// TIA Portal V19 export
FUNCTION "ALARM" : Void   // FC6, LAD
{ S7_Optimized_Access := 'TRUE' }
// stored: SetENOAutomatically false
   VAR_TEMP
      QQ : Bool;
   END_VAR
   VAR_TEMP   // added for the SCL form of the ladder/FBD networks
      _w1 : Bool;
   END_VAR
BEGIN

REGION Network 1: ALARM RESET (MASTER TO SLAVE)
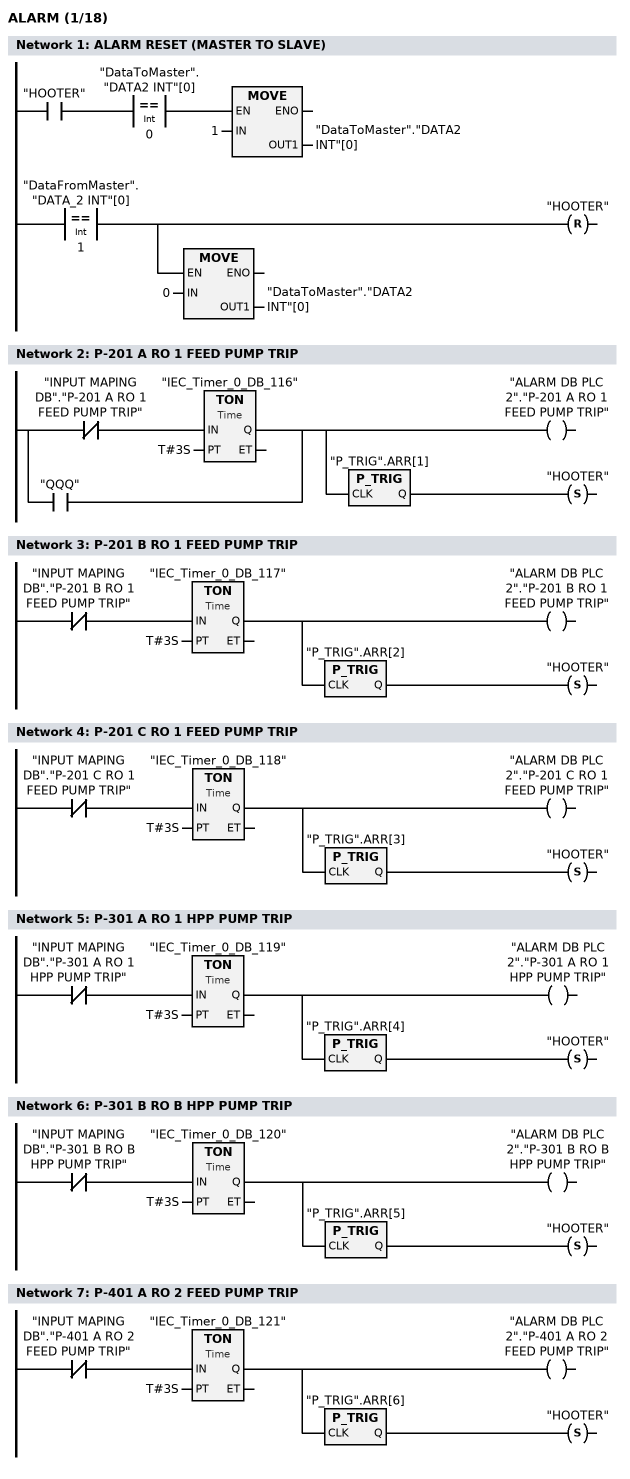
   RUNG wire#powerrail
      Contact( "HOOTER" )
      { S7_Templates := "SrcType := Int" } EQ_Contact(in1 := "DataToMaster"."DATA2 INT"[0], in2 := 0)
      Move(in := 1, out1 => "DataToMaster"."DATA2 INT"[0])
   END_RUNG
   RUNG wire#powerrail
      { S7_Templates := "SrcType := Int" } EQ_Contact(in1 := "DataFromMaster"."DATA_2 INT"[0], in2 := 1)
      wire#w1
      R_Coil( "HOOTER" )
   END_RUNG
   RUNG wire#w1
      Move(in := 0, out1 => "DataToMaster"."DATA2 INT"[0])
   END_RUNG
   // the same network as SCL:
   IF "HOOTER" AND ("DataToMaster"."DATA2 INT"[0] = 0) THEN "DataToMaster"."DATA2 INT"[0] := 1; END_IF;
   IF "DataFromMaster"."DATA_2 INT"[0] = 1 THEN
       "HOOTER" := FALSE;
       "DataToMaster"."DATA2 INT"[0] := 0;
   END_IF;
END_REGION

REGION Network 2: P-201 A RO 1 FEED PUMP TRIP
   RUNG wire#powerrail
      I_Contact( "INPUT MAPING DB"."P-201 A RO 1 FEED PUMP TRIP" )
      { S7_Templates := "time_type := Time" } "IEC_Timer_0_DB_116".TON(pt := T#3S, et =>)
      wire#w1
      Coil( "ALARM DB PLC 2"."P-201 A RO 1 FEED PUMP TRIP" )
   END_RUNG
   RUNG wire#powerrail
      Contact( "QQQ" )
   END_RUNG wire#w1
   RUNG wire#w1
      P_Trig( "P_TRIG".ARR[1] )
      S_Coil( "HOOTER" )
   END_RUNG
   // the same network as SCL:
   "IEC_Timer_0_DB_116".TON(IN := NOT "INPUT MAPING DB"."P-201 A RO 1 FEED PUMP TRIP", PT := T#3S);
   "ALARM DB PLC 2"."P-201 A RO 1 FEED PUMP TRIP" := "IEC_Timer_0_DB_116".Q OR "QQQ";
   #_w1 := "ALARM DB PLC 2"."P-201 A RO 1 FEED PUMP TRIP" AND NOT "P_TRIG".ARR[1];   // rising edge
   "P_TRIG".ARR[1] := "ALARM DB PLC 2"."P-201 A RO 1 FEED PUMP TRIP";
   IF #_w1 THEN "HOOTER" := TRUE; END_IF;
END_REGION

REGION Network 3: P-201 B RO 1 FEED PUMP TRIP
   RUNG wire#powerrail
      I_Contact( "INPUT MAPING DB"."P-201 B RO 1 FEED PUMP TRIP" )
      { S7_Templates := "time_type := Time" } "IEC_Timer_0_DB_117".TON(pt := T#3S, et =>)
      wire#w1
      Coil( "ALARM DB PLC 2"."P-201 B RO 1 FEED PUMP TRIP" )
   END_RUNG
   RUNG wire#w1
      P_Trig( "P_TRIG".ARR[2] )
      S_Coil( "HOOTER" )
   END_RUNG
   // the same network as SCL:
   "IEC_Timer_0_DB_117".TON(IN := NOT "INPUT MAPING DB"."P-201 B RO 1 FEED PUMP TRIP", PT := T#3S);
   "ALARM DB PLC 2"."P-201 B RO 1 FEED PUMP TRIP" := "IEC_Timer_0_DB_117".Q;
   #_w1 := "IEC_Timer_0_DB_117".Q AND NOT "P_TRIG".ARR[2];   // rising edge
   "P_TRIG".ARR[2] := "IEC_Timer_0_DB_117".Q;
   IF #_w1 THEN "HOOTER" := TRUE; END_IF;
END_REGION

REGION Network 4: P-201 C RO 1 FEED PUMP TRIP
   RUNG wire#powerrail
      I_Contact( "INPUT MAPING DB"."P-201 C RO 1 FEED PUMP TRIP" )
      { S7_Templates := "time_type := Time" } "IEC_Timer_0_DB_118".TON(pt := T#3S, et =>)
      wire#w1
      Coil( "ALARM DB PLC 2"."P-201 C RO 1 FEED PUMP TRIP" )
   END_RUNG
   RUNG wire#w1
      P_Trig( "P_TRIG".ARR[3] )
      S_Coil( "HOOTER" )
   END_RUNG
   // the same network as SCL:
   "IEC_Timer_0_DB_118".TON(IN := NOT "INPUT MAPING DB"."P-201 C RO 1 FEED PUMP TRIP", PT := T#3S);
   "ALARM DB PLC 2"."P-201 C RO 1 FEED PUMP TRIP" := "IEC_Timer_0_DB_118".Q;
   #_w1 := "IEC_Timer_0_DB_118".Q AND NOT "P_TRIG".ARR[3];   // rising edge
   "P_TRIG".ARR[3] := "IEC_Timer_0_DB_118".Q;
   IF #_w1 THEN "HOOTER" := TRUE; END_IF;
END_REGION

REGION Network 5: P-301 A RO 1 HPP PUMP TRIP
   RUNG wire#powerrail
      I_Contact( "INPUT MAPING DB"."P-301 A RO 1 HPP PUMP TRIP" )
      { S7_Templates := "time_type := Time" } "IEC_Timer_0_DB_119".TON(pt := T#3S, et =>)
      wire#w1
      Coil( "ALARM DB PLC 2"."P-301 A RO 1 HPP PUMP TRIP" )
   END_RUNG
   RUNG wire#w1
      P_Trig( "P_TRIG".ARR[4] )
      S_Coil( "HOOTER" )
   END_RUNG
   // the same network as SCL:
   "IEC_Timer_0_DB_119".TON(IN := NOT "INPUT MAPING DB"."P-301 A RO 1 HPP PUMP TRIP", PT := T#3S);
   "ALARM DB PLC 2"."P-301 A RO 1 HPP PUMP TRIP" := "IEC_Timer_0_DB_119".Q;
   #_w1 := "IEC_Timer_0_DB_119".Q AND NOT "P_TRIG".ARR[4];   // rising edge
   "P_TRIG".ARR[4] := "IEC_Timer_0_DB_119".Q;
   IF #_w1 THEN "HOOTER" := TRUE; END_IF;
END_REGION

REGION Network 6: P-301 B RO B HPP PUMP TRIP
   RUNG wire#powerrail
      I_Contact( "INPUT MAPING DB"."P-301 B RO B HPP PUMP TRIP" )
      { S7_Templates := "time_type := Time" } "IEC_Timer_0_DB_120".TON(pt := T#3S, et =>)
      wire#w1
      Coil( "ALARM DB PLC 2"."P-301 B RO B HPP PUMP TRIP" )
   END_RUNG
   RUNG wire#w1
      P_Trig( "P_TRIG".ARR[5] )
      S_Coil( "HOOTER" )
   END_RUNG
   // the same network as SCL:
   "IEC_Timer_0_DB_120".TON(IN := NOT "INPUT MAPING DB"."P-301 B RO B HPP PUMP TRIP", PT := T#3S);
   "ALARM DB PLC 2"."P-301 B RO B HPP PUMP TRIP" := "IEC_Timer_0_DB_120".Q;
   #_w1 := "IEC_Timer_0_DB_120".Q AND NOT "P_TRIG".ARR[5];   // rising edge
   "P_TRIG".ARR[5] := "IEC_Timer_0_DB_120".Q;
   IF #_w1 THEN "HOOTER" := TRUE; END_IF;
END_REGION

REGION Network 7: P-401 A RO 2 FEED PUMP TRIP
   RUNG wire#powerrail
      I_Contact( "INPUT MAPING DB"."P-401 A RO 2 FEED PUMP TRIP" )
      { S7_Templates := "time_type := Time" } "IEC_Timer_0_DB_121".TON(pt := T#3S, et =>)
      wire#w1
      Coil( "ALARM DB PLC 2"."P-401 A RO 2 FEED PUMP TRIP" )
   END_RUNG
   RUNG wire#w1
      P_Trig( "P_TRIG".ARR[6] )
      S_Coil( "HOOTER" )
   END_RUNG
   // the same network as SCL:
   "IEC_Timer_0_DB_121".TON(IN := NOT "INPUT MAPING DB"."P-401 A RO 2 FEED PUMP TRIP", PT := T#3S);
   "ALARM DB PLC 2"."P-401 A RO 2 FEED PUMP TRIP" := "IEC_Timer_0_DB_121".Q;
   #_w1 := "IEC_Timer_0_DB_121".Q AND NOT "P_TRIG".ARR[6];   // rising edge
   "P_TRIG".ARR[6] := "IEC_Timer_0_DB_121".Q;
   IF #_w1 THEN "HOOTER" := TRUE; END_IF;
END_REGION

REGION Network 8: P-401 B RO 2 FEED PUMP TRIP
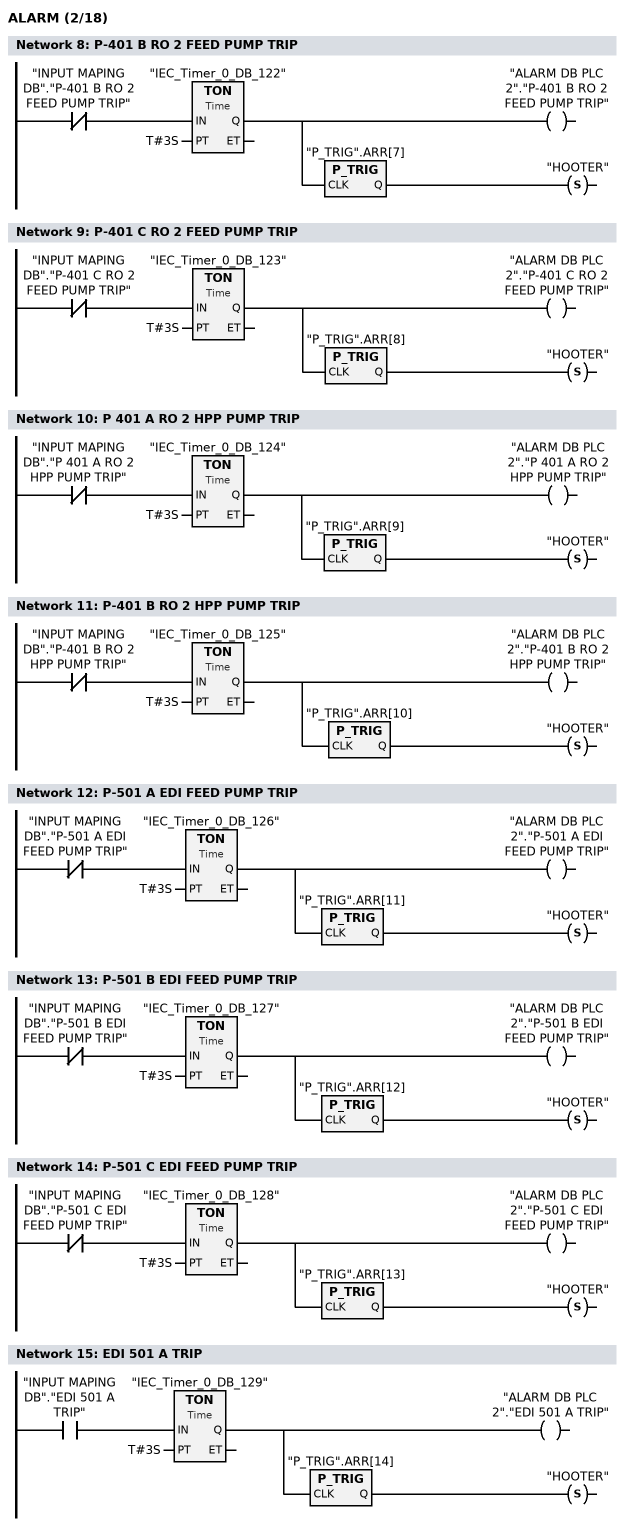
   RUNG wire#powerrail
      I_Contact( "INPUT MAPING DB"."P-401 B RO 2 FEED PUMP TRIP" )
      { S7_Templates := "time_type := Time" } "IEC_Timer_0_DB_122".TON(pt := T#3S, et =>)
      wire#w1
      Coil( "ALARM DB PLC 2"."P-401 B RO 2 FEED PUMP TRIP" )
   END_RUNG
   RUNG wire#w1
      P_Trig( "P_TRIG".ARR[7] )
      S_Coil( "HOOTER" )
   END_RUNG
   // the same network as SCL:
   "IEC_Timer_0_DB_122".TON(IN := NOT "INPUT MAPING DB"."P-401 B RO 2 FEED PUMP TRIP", PT := T#3S);
   "ALARM DB PLC 2"."P-401 B RO 2 FEED PUMP TRIP" := "IEC_Timer_0_DB_122".Q;
   #_w1 := "IEC_Timer_0_DB_122".Q AND NOT "P_TRIG".ARR[7];   // rising edge
   "P_TRIG".ARR[7] := "IEC_Timer_0_DB_122".Q;
   IF #_w1 THEN "HOOTER" := TRUE; END_IF;
END_REGION

REGION Network 9: P-401 C RO 2 FEED PUMP TRIP
   RUNG wire#powerrail
      I_Contact( "INPUT MAPING DB"."P-401 C RO 2 FEED PUMP TRIP" )
      { S7_Templates := "time_type := Time" } "IEC_Timer_0_DB_123".TON(pt := T#3S, et =>)
      wire#w1
      Coil( "ALARM DB PLC 2"."P-401 C RO 2 FEED PUMP TRIP" )
   END_RUNG
   RUNG wire#w1
      P_Trig( "P_TRIG".ARR[8] )
      S_Coil( "HOOTER" )
   END_RUNG
   // the same network as SCL:
   "IEC_Timer_0_DB_123".TON(IN := NOT "INPUT MAPING DB"."P-401 C RO 2 FEED PUMP TRIP", PT := T#3S);
   "ALARM DB PLC 2"."P-401 C RO 2 FEED PUMP TRIP" := "IEC_Timer_0_DB_123".Q;
   #_w1 := "IEC_Timer_0_DB_123".Q AND NOT "P_TRIG".ARR[8];   // rising edge
   "P_TRIG".ARR[8] := "IEC_Timer_0_DB_123".Q;
   IF #_w1 THEN "HOOTER" := TRUE; END_IF;
END_REGION

REGION Network 10: P 401 A RO 2 HPP PUMP TRIP
   RUNG wire#powerrail
      I_Contact( "INPUT MAPING DB"."P 401 A RO 2 HPP PUMP TRIP" )
      { S7_Templates := "time_type := Time" } "IEC_Timer_0_DB_124".TON(pt := T#3S, et =>)
      wire#w1
      Coil( "ALARM DB PLC 2"."P 401 A RO 2 HPP PUMP TRIP" )
   END_RUNG
   RUNG wire#w1
      P_Trig( "P_TRIG".ARR[9] )
      S_Coil( "HOOTER" )
   END_RUNG
   // the same network as SCL:
   "IEC_Timer_0_DB_124".TON(IN := NOT "INPUT MAPING DB"."P 401 A RO 2 HPP PUMP TRIP", PT := T#3S);
   "ALARM DB PLC 2"."P 401 A RO 2 HPP PUMP TRIP" := "IEC_Timer_0_DB_124".Q;
   #_w1 := "IEC_Timer_0_DB_124".Q AND NOT "P_TRIG".ARR[9];   // rising edge
   "P_TRIG".ARR[9] := "IEC_Timer_0_DB_124".Q;
   IF #_w1 THEN "HOOTER" := TRUE; END_IF;
END_REGION

REGION Network 11: P-401 B RO 2 HPP PUMP TRIP
   RUNG wire#powerrail
      I_Contact( "INPUT MAPING DB"."P-401 B RO 2 HPP PUMP TRIP" )
      { S7_Templates := "time_type := Time" } "IEC_Timer_0_DB_125".TON(pt := T#3S, et =>)
      wire#w1
      Coil( "ALARM DB PLC 2"."P-401 B RO 2 HPP PUMP TRIP" )
   END_RUNG
   RUNG wire#w1
      P_Trig( "P_TRIG".ARR[10] )
      S_Coil( "HOOTER" )
   END_RUNG
   // the same network as SCL:
   "IEC_Timer_0_DB_125".TON(IN := NOT "INPUT MAPING DB"."P-401 B RO 2 HPP PUMP TRIP", PT := T#3S);
   "ALARM DB PLC 2"."P-401 B RO 2 HPP PUMP TRIP" := "IEC_Timer_0_DB_125".Q;
   #_w1 := "IEC_Timer_0_DB_125".Q AND NOT "P_TRIG".ARR[10];   // rising edge
   "P_TRIG".ARR[10] := "IEC_Timer_0_DB_125".Q;
   IF #_w1 THEN "HOOTER" := TRUE; END_IF;
END_REGION

REGION Network 12: P-501 A EDI FEED PUMP TRIP
   RUNG wire#powerrail
      I_Contact( "INPUT MAPING DB"."P-501 A EDI FEED PUMP TRIP" )
      { S7_Templates := "time_type := Time" } "IEC_Timer_0_DB_126".TON(pt := T#3S, et =>)
      wire#w1
      Coil( "ALARM DB PLC 2"."P-501 A EDI FEED PUMP TRIP" )
   END_RUNG
   RUNG wire#w1
      P_Trig( "P_TRIG".ARR[11] )
      S_Coil( "HOOTER" )
   END_RUNG
   // the same network as SCL:
   "IEC_Timer_0_DB_126".TON(IN := NOT "INPUT MAPING DB"."P-501 A EDI FEED PUMP TRIP", PT := T#3S);
   "ALARM DB PLC 2"."P-501 A EDI FEED PUMP TRIP" := "IEC_Timer_0_DB_126".Q;
   #_w1 := "IEC_Timer_0_DB_126".Q AND NOT "P_TRIG".ARR[11];   // rising edge
   "P_TRIG".ARR[11] := "IEC_Timer_0_DB_126".Q;
   IF #_w1 THEN "HOOTER" := TRUE; END_IF;
END_REGION

REGION Network 13: P-501 B EDI FEED PUMP TRIP
   RUNG wire#powerrail
      I_Contact( "INPUT MAPING DB"."P-501 B EDI FEED PUMP TRIP" )
      { S7_Templates := "time_type := Time" } "IEC_Timer_0_DB_127".TON(pt := T#3S, et =>)
      wire#w1
      Coil( "ALARM DB PLC 2"."P-501 B EDI FEED PUMP TRIP" )
   END_RUNG
   RUNG wire#w1
      P_Trig( "P_TRIG".ARR[12] )
      S_Coil( "HOOTER" )
   END_RUNG
   // the same network as SCL:
   "IEC_Timer_0_DB_127".TON(IN := NOT "INPUT MAPING DB"."P-501 B EDI FEED PUMP TRIP", PT := T#3S);
   "ALARM DB PLC 2"."P-501 B EDI FEED PUMP TRIP" := "IEC_Timer_0_DB_127".Q;
   #_w1 := "IEC_Timer_0_DB_127".Q AND NOT "P_TRIG".ARR[12];   // rising edge
   "P_TRIG".ARR[12] := "IEC_Timer_0_DB_127".Q;
   IF #_w1 THEN "HOOTER" := TRUE; END_IF;
END_REGION

REGION Network 14: P-501 C EDI FEED PUMP TRIP
   RUNG wire#powerrail
      I_Contact( "INPUT MAPING DB"."P-501 C EDI FEED PUMP TRIP" )
      { S7_Templates := "time_type := Time" } "IEC_Timer_0_DB_128".TON(pt := T#3S, et =>)
      wire#w1
      Coil( "ALARM DB PLC 2"."P-501 C EDI FEED PUMP TRIP" )
   END_RUNG
   RUNG wire#w1
      P_Trig( "P_TRIG".ARR[13] )
      S_Coil( "HOOTER" )
   END_RUNG
   // the same network as SCL:
   "IEC_Timer_0_DB_128".TON(IN := NOT "INPUT MAPING DB"."P-501 C EDI FEED PUMP TRIP", PT := T#3S);
   "ALARM DB PLC 2"."P-501 C EDI FEED PUMP TRIP" := "IEC_Timer_0_DB_128".Q;
   #_w1 := "IEC_Timer_0_DB_128".Q AND NOT "P_TRIG".ARR[13];   // rising edge
   "P_TRIG".ARR[13] := "IEC_Timer_0_DB_128".Q;
   IF #_w1 THEN "HOOTER" := TRUE; END_IF;
END_REGION

REGION Network 15: EDI 501 A TRIP
   RUNG wire#powerrail
      Contact( "INPUT MAPING DB"."EDI 501 A TRIP" )
      { S7_Templates := "time_type := Time" } "IEC_Timer_0_DB_129".TON(pt := T#3S, et =>)
      wire#w1
      Coil( "ALARM DB PLC 2"."EDI 501 A TRIP" )
   END_RUNG
   RUNG wire#w1
      P_Trig( "P_TRIG".ARR[14] )
      S_Coil( "HOOTER" )
   END_RUNG
   // the same network as SCL:
   "IEC_Timer_0_DB_129".TON(IN := "INPUT MAPING DB"."EDI 501 A TRIP", PT := T#3S);
   "ALARM DB PLC 2"."EDI 501 A TRIP" := "IEC_Timer_0_DB_129".Q;
   #_w1 := "IEC_Timer_0_DB_129".Q AND NOT "P_TRIG".ARR[14];   // rising edge
   "P_TRIG".ARR[14] := "IEC_Timer_0_DB_129".Q;
   IF #_w1 THEN "HOOTER" := TRUE; END_IF;
END_REGION

REGION Network 16: EDI 501 B TRIP
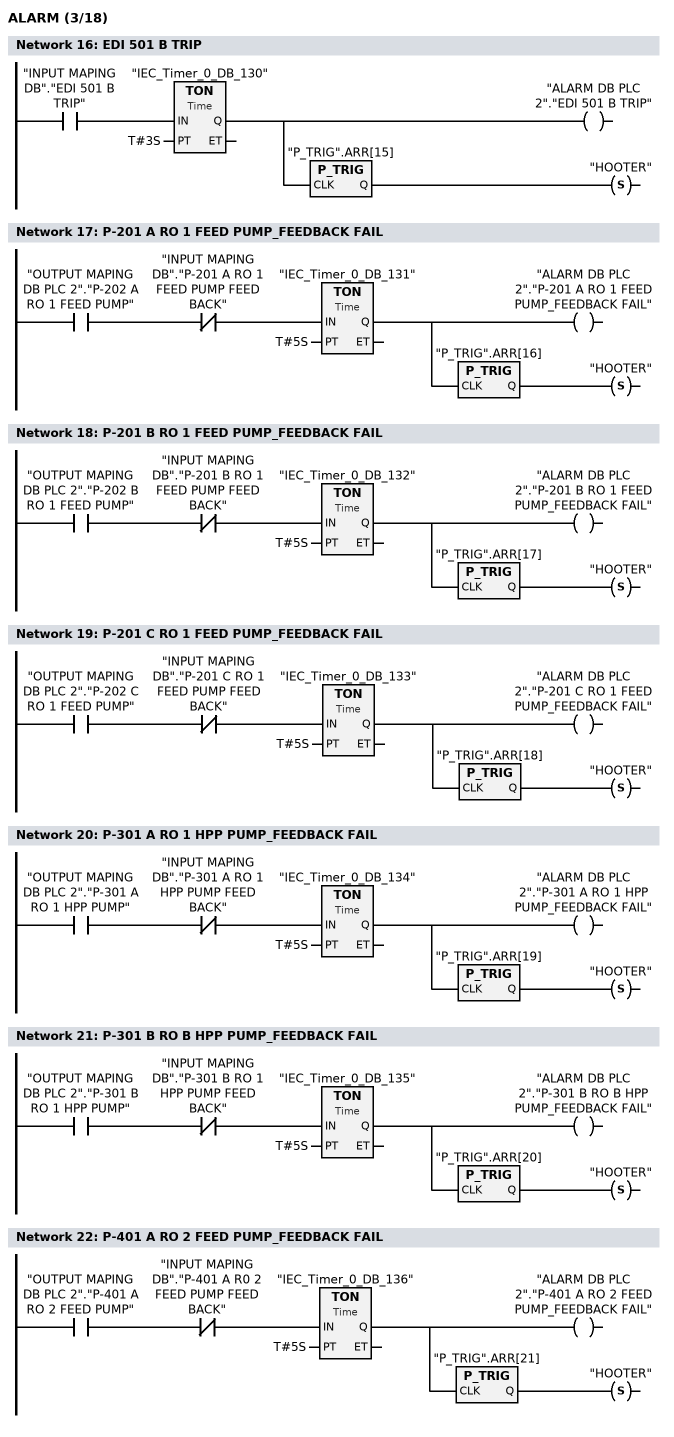
   RUNG wire#powerrail
      Contact( "INPUT MAPING DB"."EDI 501 B TRIP" )
      { S7_Templates := "time_type := Time" } "IEC_Timer_0_DB_130".TON(pt := T#3S, et =>)
      wire#w1
      Coil( "ALARM DB PLC 2"."EDI 501 B TRIP" )
   END_RUNG
   RUNG wire#w1
      P_Trig( "P_TRIG".ARR[15] )
      S_Coil( "HOOTER" )
   END_RUNG
   // the same network as SCL:
   "IEC_Timer_0_DB_130".TON(IN := "INPUT MAPING DB"."EDI 501 B TRIP", PT := T#3S);
   "ALARM DB PLC 2"."EDI 501 B TRIP" := "IEC_Timer_0_DB_130".Q;
   #_w1 := "IEC_Timer_0_DB_130".Q AND NOT "P_TRIG".ARR[15];   // rising edge
   "P_TRIG".ARR[15] := "IEC_Timer_0_DB_130".Q;
   IF #_w1 THEN "HOOTER" := TRUE; END_IF;
END_REGION

REGION Network 17: P-201 A RO 1 FEED PUMP_FEEDBACK FAIL
   RUNG wire#powerrail
      Contact( "OUTPUT MAPING DB PLC 2"."P-202 A RO 1 FEED PUMP" )
      I_Contact( "INPUT MAPING DB"."P-201 A RO 1 FEED PUMP FEED BACK" )
      { S7_Templates := "time_type := Time" } "IEC_Timer_0_DB_131".TON(pt := T#5S, et =>)
      wire#w1
      Coil( "ALARM DB PLC 2"."P-201 A RO 1 FEED PUMP_FEEDBACK FAIL" )
   END_RUNG
   RUNG wire#w1
      P_Trig( "P_TRIG".ARR[16] )
      S_Coil( "HOOTER" )
   END_RUNG
   // the same network as SCL:
   "IEC_Timer_0_DB_131".TON(IN := "OUTPUT MAPING DB PLC 2"."P-202 A RO 1 FEED PUMP" AND NOT "INPUT MAPING DB"."P-201 A RO 1 FEED PUMP FEED BACK",
                           PT := T#5S);
   "ALARM DB PLC 2"."P-201 A RO 1 FEED PUMP_FEEDBACK FAIL" := "IEC_Timer_0_DB_131".Q;
   #_w1 := "IEC_Timer_0_DB_131".Q AND NOT "P_TRIG".ARR[16];   // rising edge
   "P_TRIG".ARR[16] := "IEC_Timer_0_DB_131".Q;
   IF #_w1 THEN "HOOTER" := TRUE; END_IF;
END_REGION

REGION Network 18: P-201 B RO 1 FEED PUMP_FEEDBACK FAIL
   RUNG wire#powerrail
      Contact( "OUTPUT MAPING DB PLC 2"."P-202 B RO 1 FEED PUMP" )
      I_Contact( "INPUT MAPING DB"."P-201 B RO 1 FEED PUMP FEED BACK" )
      { S7_Templates := "time_type := Time" } "IEC_Timer_0_DB_132".TON(pt := T#5S, et =>)
      wire#w1
      Coil( "ALARM DB PLC 2"."P-201 B RO 1 FEED PUMP_FEEDBACK FAIL" )
   END_RUNG
   RUNG wire#w1
      P_Trig( "P_TRIG".ARR[17] )
      S_Coil( "HOOTER" )
   END_RUNG
   // the same network as SCL:
   "IEC_Timer_0_DB_132".TON(IN := "OUTPUT MAPING DB PLC 2"."P-202 B RO 1 FEED PUMP" AND NOT "INPUT MAPING DB"."P-201 B RO 1 FEED PUMP FEED BACK",
                           PT := T#5S);
   "ALARM DB PLC 2"."P-201 B RO 1 FEED PUMP_FEEDBACK FAIL" := "IEC_Timer_0_DB_132".Q;
   #_w1 := "IEC_Timer_0_DB_132".Q AND NOT "P_TRIG".ARR[17];   // rising edge
   "P_TRIG".ARR[17] := "IEC_Timer_0_DB_132".Q;
   IF #_w1 THEN "HOOTER" := TRUE; END_IF;
END_REGION

REGION Network 19: P-201 C RO 1 FEED PUMP_FEEDBACK FAIL
   RUNG wire#powerrail
      Contact( "OUTPUT MAPING DB PLC 2"."P-202 C RO 1 FEED PUMP" )
      I_Contact( "INPUT MAPING DB"."P-201 C RO 1 FEED PUMP FEED BACK" )
      { S7_Templates := "time_type := Time" } "IEC_Timer_0_DB_133".TON(pt := T#5S, et =>)
      wire#w1
      Coil( "ALARM DB PLC 2"."P-201 C RO 1 FEED PUMP_FEEDBACK FAIL" )
   END_RUNG
   RUNG wire#w1
      P_Trig( "P_TRIG".ARR[18] )
      S_Coil( "HOOTER" )
   END_RUNG
   // the same network as SCL:
   "IEC_Timer_0_DB_133".TON(IN := "OUTPUT MAPING DB PLC 2"."P-202 C RO 1 FEED PUMP" AND NOT "INPUT MAPING DB"."P-201 C RO 1 FEED PUMP FEED BACK",
                           PT := T#5S);
   "ALARM DB PLC 2"."P-201 C RO 1 FEED PUMP_FEEDBACK FAIL" := "IEC_Timer_0_DB_133".Q;
   #_w1 := "IEC_Timer_0_DB_133".Q AND NOT "P_TRIG".ARR[18];   // rising edge
   "P_TRIG".ARR[18] := "IEC_Timer_0_DB_133".Q;
   IF #_w1 THEN "HOOTER" := TRUE; END_IF;
END_REGION

REGION Network 20: P-301 A RO 1 HPP PUMP_FEEDBACK FAIL
   RUNG wire#powerrail
      Contact( "OUTPUT MAPING DB PLC 2"."P-301 A RO 1 HPP PUMP" )
      I_Contact( "INPUT MAPING DB"."P-301 A RO 1 HPP PUMP FEED BACK" )
      { S7_Templates := "time_type := Time" } "IEC_Timer_0_DB_134".TON(pt := T#5S, et =>)
      wire#w1
      Coil( "ALARM DB PLC 2"."P-301 A RO 1 HPP PUMP_FEEDBACK FAIL" )
   END_RUNG
   RUNG wire#w1
      P_Trig( "P_TRIG".ARR[19] )
      S_Coil( "HOOTER" )
   END_RUNG
   // the same network as SCL:
   "IEC_Timer_0_DB_134".TON(IN := "OUTPUT MAPING DB PLC 2"."P-301 A RO 1 HPP PUMP" AND NOT "INPUT MAPING DB"."P-301 A RO 1 HPP PUMP FEED BACK",
                           PT := T#5S);
   "ALARM DB PLC 2"."P-301 A RO 1 HPP PUMP_FEEDBACK FAIL" := "IEC_Timer_0_DB_134".Q;
   #_w1 := "IEC_Timer_0_DB_134".Q AND NOT "P_TRIG".ARR[19];   // rising edge
   "P_TRIG".ARR[19] := "IEC_Timer_0_DB_134".Q;
   IF #_w1 THEN "HOOTER" := TRUE; END_IF;
END_REGION

REGION Network 21: P-301 B RO B HPP PUMP_FEEDBACK FAIL
   RUNG wire#powerrail
      Contact( "OUTPUT MAPING DB PLC 2"."P-301 B RO 1 HPP PUMP" )
      I_Contact( "INPUT MAPING DB"."P-301 B RO 1 HPP PUMP FEED BACK" )
      { S7_Templates := "time_type := Time" } "IEC_Timer_0_DB_135".TON(pt := T#5S, et =>)
      wire#w1
      Coil( "ALARM DB PLC 2"."P-301 B RO B HPP PUMP_FEEDBACK FAIL" )
   END_RUNG
   RUNG wire#w1
      P_Trig( "P_TRIG".ARR[20] )
      S_Coil( "HOOTER" )
   END_RUNG
   // the same network as SCL:
   "IEC_Timer_0_DB_135".TON(IN := "OUTPUT MAPING DB PLC 2"."P-301 B RO 1 HPP PUMP" AND NOT "INPUT MAPING DB"."P-301 B RO 1 HPP PUMP FEED BACK",
                           PT := T#5S);
   "ALARM DB PLC 2"."P-301 B RO B HPP PUMP_FEEDBACK FAIL" := "IEC_Timer_0_DB_135".Q;
   #_w1 := "IEC_Timer_0_DB_135".Q AND NOT "P_TRIG".ARR[20];   // rising edge
   "P_TRIG".ARR[20] := "IEC_Timer_0_DB_135".Q;
   IF #_w1 THEN "HOOTER" := TRUE; END_IF;
END_REGION

REGION Network 22: P-401 A RO 2 FEED PUMP_FEEDBACK FAIL
   RUNG wire#powerrail
      Contact( "OUTPUT MAPING DB PLC 2"."P-401 A RO 2 FEED PUMP" )
      I_Contact( "INPUT MAPING DB"."P-401 A R0 2 FEED PUMP FEED BACK" )
      { S7_Templates := "time_type := Time" } "IEC_Timer_0_DB_136".TON(pt := T#5S, et =>)
      wire#w1
      Coil( "ALARM DB PLC 2"."P-401 A RO 2 FEED PUMP_FEEDBACK FAIL" )
   END_RUNG
   RUNG wire#w1
      P_Trig( "P_TRIG".ARR[21] )
      S_Coil( "HOOTER" )
   END_RUNG
   // the same network as SCL:
   "IEC_Timer_0_DB_136".TON(IN := "OUTPUT MAPING DB PLC 2"."P-401 A RO 2 FEED PUMP" AND NOT "INPUT MAPING DB"."P-401 A R0 2 FEED PUMP FEED BACK",
                           PT := T#5S);
   "ALARM DB PLC 2"."P-401 A RO 2 FEED PUMP_FEEDBACK FAIL" := "IEC_Timer_0_DB_136".Q;
   #_w1 := "IEC_Timer_0_DB_136".Q AND NOT "P_TRIG".ARR[21];   // rising edge
   "P_TRIG".ARR[21] := "IEC_Timer_0_DB_136".Q;
   IF #_w1 THEN "HOOTER" := TRUE; END_IF;
END_REGION

REGION Network 23: P-401 B RO 2 FEED PUMP_FEEDBACK FAIL
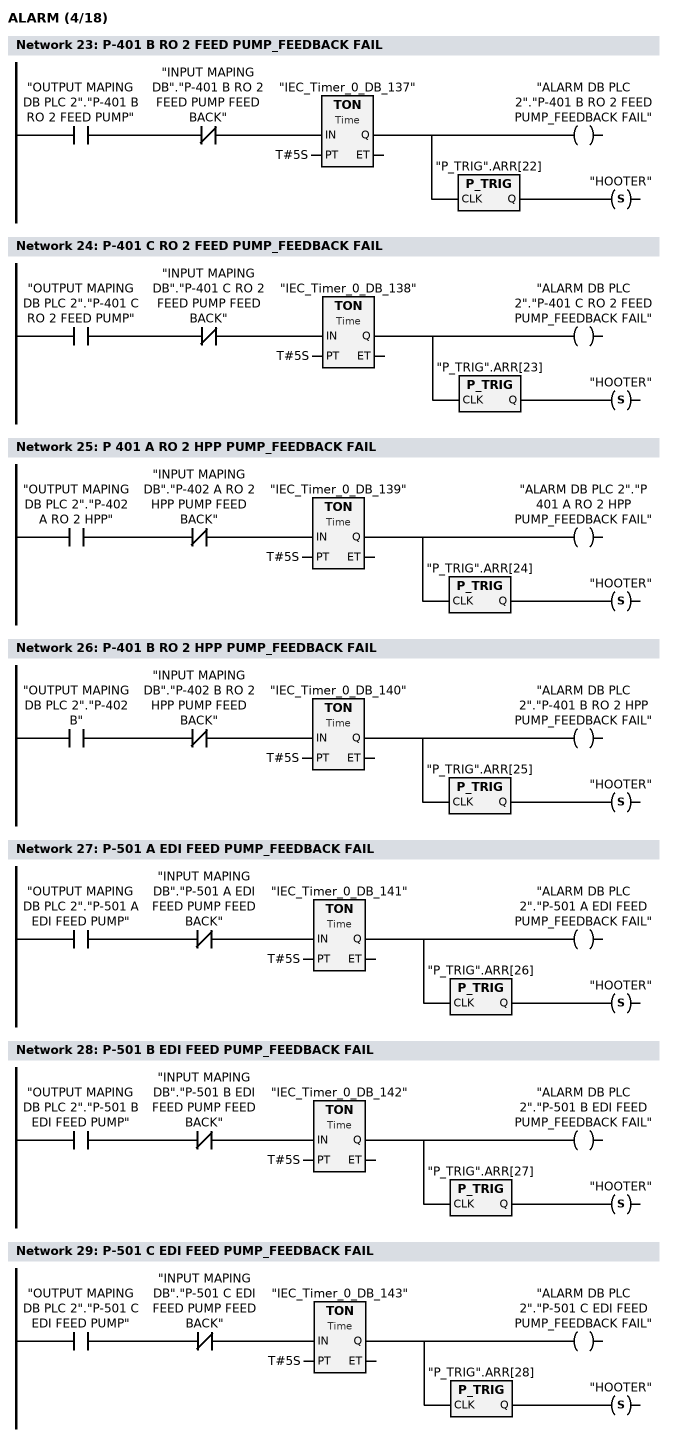
   RUNG wire#powerrail
      Contact( "OUTPUT MAPING DB PLC 2"."P-401 B RO 2 FEED PUMP" )
      I_Contact( "INPUT MAPING DB"."P-401 B RO 2 FEED PUMP FEED BACK" )
      { S7_Templates := "time_type := Time" } "IEC_Timer_0_DB_137".TON(pt := T#5S, et =>)
      wire#w1
      Coil( "ALARM DB PLC 2"."P-401 B RO 2 FEED PUMP_FEEDBACK FAIL" )
   END_RUNG
   RUNG wire#w1
      P_Trig( "P_TRIG".ARR[22] )
      S_Coil( "HOOTER" )
   END_RUNG
   // the same network as SCL:
   "IEC_Timer_0_DB_137".TON(IN := "OUTPUT MAPING DB PLC 2"."P-401 B RO 2 FEED PUMP" AND NOT "INPUT MAPING DB"."P-401 B RO 2 FEED PUMP FEED BACK",
                           PT := T#5S);
   "ALARM DB PLC 2"."P-401 B RO 2 FEED PUMP_FEEDBACK FAIL" := "IEC_Timer_0_DB_137".Q;
   #_w1 := "IEC_Timer_0_DB_137".Q AND NOT "P_TRIG".ARR[22];   // rising edge
   "P_TRIG".ARR[22] := "IEC_Timer_0_DB_137".Q;
   IF #_w1 THEN "HOOTER" := TRUE; END_IF;
END_REGION

REGION Network 24: P-401 C RO 2 FEED PUMP_FEEDBACK FAIL
   RUNG wire#powerrail
      Contact( "OUTPUT MAPING DB PLC 2"."P-401 C RO 2 FEED PUMP" )
      I_Contact( "INPUT MAPING DB"."P-401 C RO 2 FEED PUMP FEED BACK" )
      { S7_Templates := "time_type := Time" } "IEC_Timer_0_DB_138".TON(pt := T#5S, et =>)
      wire#w1
      Coil( "ALARM DB PLC 2"."P-401 C RO 2 FEED PUMP_FEEDBACK FAIL" )
   END_RUNG
   RUNG wire#w1
      P_Trig( "P_TRIG".ARR[23] )
      S_Coil( "HOOTER" )
   END_RUNG
   // the same network as SCL:
   "IEC_Timer_0_DB_138".TON(IN := "OUTPUT MAPING DB PLC 2"."P-401 C RO 2 FEED PUMP" AND NOT "INPUT MAPING DB"."P-401 C RO 2 FEED PUMP FEED BACK",
                           PT := T#5S);
   "ALARM DB PLC 2"."P-401 C RO 2 FEED PUMP_FEEDBACK FAIL" := "IEC_Timer_0_DB_138".Q;
   #_w1 := "IEC_Timer_0_DB_138".Q AND NOT "P_TRIG".ARR[23];   // rising edge
   "P_TRIG".ARR[23] := "IEC_Timer_0_DB_138".Q;
   IF #_w1 THEN "HOOTER" := TRUE; END_IF;
END_REGION

REGION Network 25: P 401 A RO 2 HPP PUMP_FEEDBACK FAIL
   RUNG wire#powerrail
      Contact( "OUTPUT MAPING DB PLC 2"."P-402  A RO 2 HPP" )
      I_Contact( "INPUT MAPING DB"."P-402 A RO 2 HPP PUMP FEED BACK" )
      { S7_Templates := "time_type := Time" } "IEC_Timer_0_DB_139".TON(pt := T#5S, et =>)
      wire#w1
      Coil( "ALARM DB PLC 2"."P 401 A RO 2 HPP PUMP_FEEDBACK FAIL" )
   END_RUNG
   RUNG wire#w1
      P_Trig( "P_TRIG".ARR[24] )
      S_Coil( "HOOTER" )
   END_RUNG
   // the same network as SCL:
   "IEC_Timer_0_DB_139".TON(IN := "OUTPUT MAPING DB PLC 2"."P-402  A RO 2 HPP" AND NOT "INPUT MAPING DB"."P-402 A RO 2 HPP PUMP FEED BACK",
                           PT := T#5S);
   "ALARM DB PLC 2"."P 401 A RO 2 HPP PUMP_FEEDBACK FAIL" := "IEC_Timer_0_DB_139".Q;
   #_w1 := "IEC_Timer_0_DB_139".Q AND NOT "P_TRIG".ARR[24];   // rising edge
   "P_TRIG".ARR[24] := "IEC_Timer_0_DB_139".Q;
   IF #_w1 THEN "HOOTER" := TRUE; END_IF;
END_REGION

REGION Network 26: P-401 B RO 2 HPP PUMP_FEEDBACK FAIL
   RUNG wire#powerrail
      Contact( "OUTPUT MAPING DB PLC 2"."P-402 B" )
      I_Contact( "INPUT MAPING DB"."P-402 B RO 2 HPP PUMP FEED BACK" )
      { S7_Templates := "time_type := Time" } "IEC_Timer_0_DB_140".TON(pt := T#5S, et =>)
      wire#w1
      Coil( "ALARM DB PLC 2"."P-401 B RO 2 HPP PUMP_FEEDBACK FAIL" )
   END_RUNG
   RUNG wire#w1
      P_Trig( "P_TRIG".ARR[25] )
      S_Coil( "HOOTER" )
   END_RUNG
   // the same network as SCL:
   "IEC_Timer_0_DB_140".TON(IN := "OUTPUT MAPING DB PLC 2"."P-402 B" AND NOT "INPUT MAPING DB"."P-402 B RO 2 HPP PUMP FEED BACK",
                           PT := T#5S);
   "ALARM DB PLC 2"."P-401 B RO 2 HPP PUMP_FEEDBACK FAIL" := "IEC_Timer_0_DB_140".Q;
   #_w1 := "IEC_Timer_0_DB_140".Q AND NOT "P_TRIG".ARR[25];   // rising edge
   "P_TRIG".ARR[25] := "IEC_Timer_0_DB_140".Q;
   IF #_w1 THEN "HOOTER" := TRUE; END_IF;
END_REGION

REGION Network 27: P-501 A EDI FEED PUMP_FEEDBACK FAIL
   RUNG wire#powerrail
      Contact( "OUTPUT MAPING DB PLC 2"."P-501 A EDI FEED PUMP" )
      I_Contact( "INPUT MAPING DB"."P-501 A EDI FEED PUMP FEED BACK" )
      { S7_Templates := "time_type := Time" } "IEC_Timer_0_DB_141".TON(pt := T#5S, et =>)
      wire#w1
      Coil( "ALARM DB PLC 2"."P-501 A EDI FEED PUMP_FEEDBACK FAIL" )
   END_RUNG
   RUNG wire#w1
      P_Trig( "P_TRIG".ARR[26] )
      S_Coil( "HOOTER" )
   END_RUNG
   // the same network as SCL:
   "IEC_Timer_0_DB_141".TON(IN := "OUTPUT MAPING DB PLC 2"."P-501 A EDI FEED PUMP" AND NOT "INPUT MAPING DB"."P-501 A EDI FEED PUMP FEED BACK",
                           PT := T#5S);
   "ALARM DB PLC 2"."P-501 A EDI FEED PUMP_FEEDBACK FAIL" := "IEC_Timer_0_DB_141".Q;
   #_w1 := "IEC_Timer_0_DB_141".Q AND NOT "P_TRIG".ARR[26];   // rising edge
   "P_TRIG".ARR[26] := "IEC_Timer_0_DB_141".Q;
   IF #_w1 THEN "HOOTER" := TRUE; END_IF;
END_REGION

REGION Network 28: P-501 B EDI FEED PUMP_FEEDBACK FAIL
   RUNG wire#powerrail
      Contact( "OUTPUT MAPING DB PLC 2"."P-501 B EDI FEED PUMP" )
      I_Contact( "INPUT MAPING DB"."P-501 B EDI FEED PUMP FEED BACK" )
      { S7_Templates := "time_type := Time" } "IEC_Timer_0_DB_142".TON(pt := T#5S, et =>)
      wire#w1
      Coil( "ALARM DB PLC 2"."P-501 B EDI FEED PUMP_FEEDBACK FAIL" )
   END_RUNG
   RUNG wire#w1
      P_Trig( "P_TRIG".ARR[27] )
      S_Coil( "HOOTER" )
   END_RUNG
   // the same network as SCL:
   "IEC_Timer_0_DB_142".TON(IN := "OUTPUT MAPING DB PLC 2"."P-501 B EDI FEED PUMP" AND NOT "INPUT MAPING DB"."P-501 B EDI FEED PUMP FEED BACK",
                           PT := T#5S);
   "ALARM DB PLC 2"."P-501 B EDI FEED PUMP_FEEDBACK FAIL" := "IEC_Timer_0_DB_142".Q;
   #_w1 := "IEC_Timer_0_DB_142".Q AND NOT "P_TRIG".ARR[27];   // rising edge
   "P_TRIG".ARR[27] := "IEC_Timer_0_DB_142".Q;
   IF #_w1 THEN "HOOTER" := TRUE; END_IF;
END_REGION

REGION Network 29: P-501 C EDI FEED PUMP_FEEDBACK FAIL
   RUNG wire#powerrail
      Contact( "OUTPUT MAPING DB PLC 2"."P-501 C EDI FEED PUMP" )
      I_Contact( "INPUT MAPING DB"."P-501 C EDI FEED PUMP FEED BACK" )
      { S7_Templates := "time_type := Time" } "IEC_Timer_0_DB_143".TON(pt := T#5S, et =>)
      wire#w1
      Coil( "ALARM DB PLC 2"."P-501 C EDI FEED PUMP_FEEDBACK FAIL" )
   END_RUNG
   RUNG wire#w1
      P_Trig( "P_TRIG".ARR[28] )
      S_Coil( "HOOTER" )
   END_RUNG
   // the same network as SCL:
   "IEC_Timer_0_DB_143".TON(IN := "OUTPUT MAPING DB PLC 2"."P-501 C EDI FEED PUMP" AND NOT "INPUT MAPING DB"."P-501 C EDI FEED PUMP FEED BACK",
                           PT := T#5S);
   "ALARM DB PLC 2"."P-501 C EDI FEED PUMP_FEEDBACK FAIL" := "IEC_Timer_0_DB_143".Q;
   #_w1 := "IEC_Timer_0_DB_143".Q AND NOT "P_TRIG".ARR[28];   // rising edge
   "P_TRIG".ARR[28] := "IEC_Timer_0_DB_143".Q;
   IF #_w1 THEN "HOOTER" := TRUE; END_IF;
END_REGION

REGION Network 30: EDI 501 A _FEEDBACK FAIL
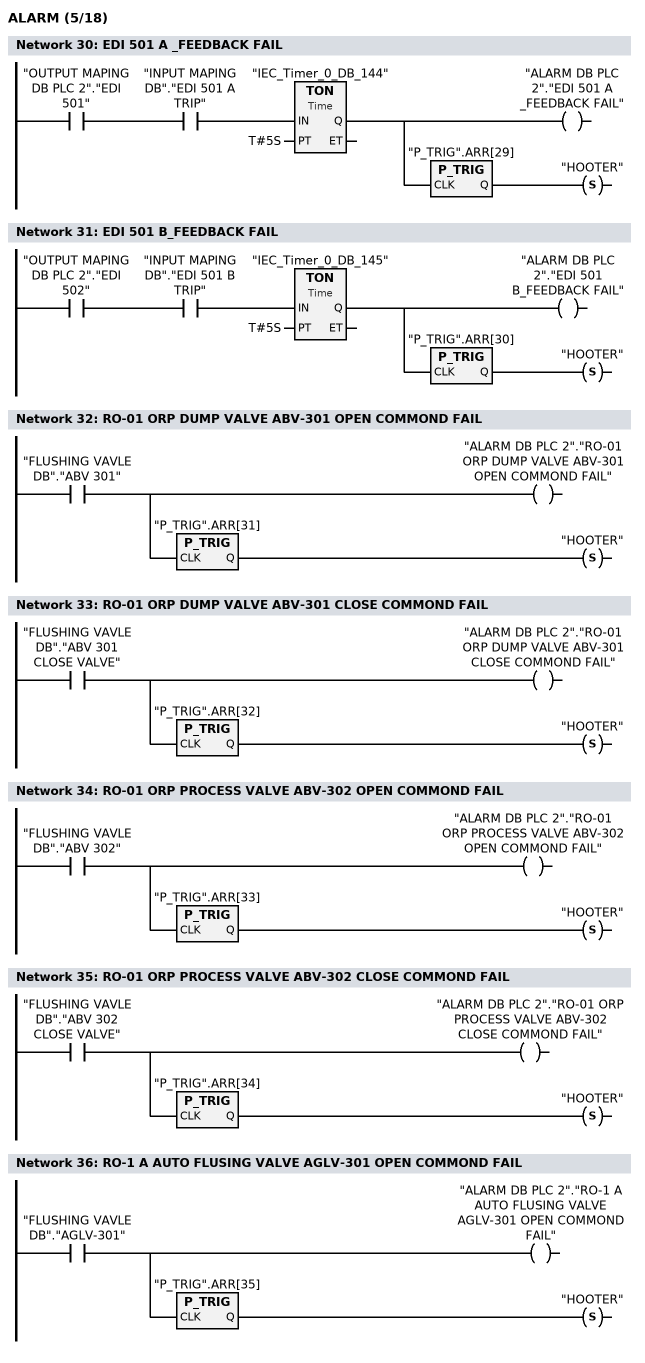
   RUNG wire#powerrail
      Contact( "OUTPUT MAPING DB PLC 2"."EDI 501" )
      Contact( "INPUT MAPING DB"."EDI 501 A TRIP" )
      { S7_Templates := "time_type := Time" } "IEC_Timer_0_DB_144".TON(pt := T#5S, et =>)
      wire#w1
      Coil( "ALARM DB PLC 2"."EDI 501 A _FEEDBACK FAIL" )
   END_RUNG
   RUNG wire#w1
      P_Trig( "P_TRIG".ARR[29] )
      S_Coil( "HOOTER" )
   END_RUNG
   // the same network as SCL:
   "IEC_Timer_0_DB_144".TON(IN := "OUTPUT MAPING DB PLC 2"."EDI 501" AND "INPUT MAPING DB"."EDI 501 A TRIP",
                           PT := T#5S);
   "ALARM DB PLC 2"."EDI 501 A _FEEDBACK FAIL" := "IEC_Timer_0_DB_144".Q;
   #_w1 := "IEC_Timer_0_DB_144".Q AND NOT "P_TRIG".ARR[29];   // rising edge
   "P_TRIG".ARR[29] := "IEC_Timer_0_DB_144".Q;
   IF #_w1 THEN "HOOTER" := TRUE; END_IF;
END_REGION

REGION Network 31: EDI 501 B_FEEDBACK FAIL
   RUNG wire#powerrail
      Contact( "OUTPUT MAPING DB PLC 2"."EDI 502" )
      Contact( "INPUT MAPING DB"."EDI 501 B TRIP" )
      { S7_Templates := "time_type := Time" } "IEC_Timer_0_DB_145".TON(pt := T#5S, et =>)
      wire#w1
      Coil( "ALARM DB PLC 2"."EDI 501 B_FEEDBACK FAIL" )
   END_RUNG
   RUNG wire#w1
      P_Trig( "P_TRIG".ARR[30] )
      S_Coil( "HOOTER" )
   END_RUNG
   // the same network as SCL:
   "IEC_Timer_0_DB_145".TON(IN := "OUTPUT MAPING DB PLC 2"."EDI 502" AND "INPUT MAPING DB"."EDI 501 B TRIP",
                           PT := T#5S);
   "ALARM DB PLC 2"."EDI 501 B_FEEDBACK FAIL" := "IEC_Timer_0_DB_145".Q;
   #_w1 := "IEC_Timer_0_DB_145".Q AND NOT "P_TRIG".ARR[30];   // rising edge
   "P_TRIG".ARR[30] := "IEC_Timer_0_DB_145".Q;
   IF #_w1 THEN "HOOTER" := TRUE; END_IF;
END_REGION

REGION Network 32: RO-01 ORP DUMP VALVE ABV-301 OPEN COMMOND FAIL
   RUNG wire#powerrail
      Contact( "FLUSHING VAVLE DB"."ABV 301" )
      wire#w1
      Coil( "ALARM DB PLC 2"."RO-01 ORP DUMP VALVE ABV-301 OPEN COMMOND FAIL" )
   END_RUNG
   RUNG wire#w1
      P_Trig( "P_TRIG".ARR[31] )
      S_Coil( "HOOTER" )
   END_RUNG
   // the same network as SCL:
   "ALARM DB PLC 2"."RO-01 ORP DUMP VALVE ABV-301 OPEN COMMOND FAIL" := "FLUSHING VAVLE DB"."ABV 301";
   #_w1 := "FLUSHING VAVLE DB"."ABV 301" AND NOT "P_TRIG".ARR[31];   // rising edge
   "P_TRIG".ARR[31] := "FLUSHING VAVLE DB"."ABV 301";
   IF #_w1 THEN "HOOTER" := TRUE; END_IF;
END_REGION

REGION Network 33: RO-01 ORP DUMP VALVE ABV-301 CLOSE COMMOND FAIL
   RUNG wire#powerrail
      Contact( "FLUSHING VAVLE DB"."ABV 301 CLOSE VALVE" )
      wire#w1
      Coil( "ALARM DB PLC 2"."RO-01 ORP DUMP VALVE ABV-301 CLOSE COMMOND FAIL" )
   END_RUNG
   RUNG wire#w1
      P_Trig( "P_TRIG".ARR[32] )
      S_Coil( "HOOTER" )
   END_RUNG
   // the same network as SCL:
   "ALARM DB PLC 2"."RO-01 ORP DUMP VALVE ABV-301 CLOSE COMMOND FAIL" := "FLUSHING VAVLE DB"."ABV 301 CLOSE VALVE";
   #_w1 := "FLUSHING VAVLE DB"."ABV 301 CLOSE VALVE" AND NOT "P_TRIG".ARR[32];   // rising edge
   "P_TRIG".ARR[32] := "FLUSHING VAVLE DB"."ABV 301 CLOSE VALVE";
   IF #_w1 THEN "HOOTER" := TRUE; END_IF;
END_REGION

REGION Network 34: RO-01 ORP PROCESS VALVE ABV-302 OPEN COMMOND FAIL
   RUNG wire#powerrail
      Contact( "FLUSHING VAVLE DB"."ABV 302" )
      wire#w1
      Coil( "ALARM DB PLC 2"."RO-01 ORP PROCESS VALVE ABV-302 OPEN COMMOND FAIL" )
   END_RUNG
   RUNG wire#w1
      P_Trig( "P_TRIG".ARR[33] )
      S_Coil( "HOOTER" )
   END_RUNG
   // the same network as SCL:
   "ALARM DB PLC 2"."RO-01 ORP PROCESS VALVE ABV-302 OPEN COMMOND FAIL" := "FLUSHING VAVLE DB"."ABV 302";
   #_w1 := "FLUSHING VAVLE DB"."ABV 302" AND NOT "P_TRIG".ARR[33];   // rising edge
   "P_TRIG".ARR[33] := "FLUSHING VAVLE DB"."ABV 302";
   IF #_w1 THEN "HOOTER" := TRUE; END_IF;
END_REGION

REGION Network 35: RO-01 ORP PROCESS VALVE ABV-302 CLOSE COMMOND FAIL
   RUNG wire#powerrail
      Contact( "FLUSHING VAVLE DB"."ABV 302 CLOSE VALVE" )
      wire#w1
      Coil( "ALARM DB PLC 2"."RO-01 ORP PROCESS VALVE ABV-302 CLOSE COMMOND FAIL" )
   END_RUNG
   RUNG wire#w1
      P_Trig( "P_TRIG".ARR[34] )
      S_Coil( "HOOTER" )
   END_RUNG
   // the same network as SCL:
   "ALARM DB PLC 2"."RO-01 ORP PROCESS VALVE ABV-302 CLOSE COMMOND FAIL" := "FLUSHING VAVLE DB"."ABV 302 CLOSE VALVE";
   #_w1 := "FLUSHING VAVLE DB"."ABV 302 CLOSE VALVE" AND NOT "P_TRIG".ARR[34];   // rising edge
   "P_TRIG".ARR[34] := "FLUSHING VAVLE DB"."ABV 302 CLOSE VALVE";
   IF #_w1 THEN "HOOTER" := TRUE; END_IF;
END_REGION

REGION Network 36: RO-1 A AUTO FLUSING VALVE AGLV-301 OPEN COMMOND FAIL
   RUNG wire#powerrail
      Contact( "FLUSHING VAVLE DB"."AGLV-301" )
      wire#w1
      Coil( "ALARM DB PLC 2"."RO-1 A AUTO FLUSING VALVE AGLV-301 OPEN COMMOND FAIL" )
   END_RUNG
   RUNG wire#w1
      P_Trig( "P_TRIG".ARR[35] )
      S_Coil( "HOOTER" )
   END_RUNG
   // the same network as SCL:
   "ALARM DB PLC 2"."RO-1 A AUTO FLUSING VALVE AGLV-301 OPEN COMMOND FAIL" := "FLUSHING VAVLE DB"."AGLV-301";
   #_w1 := "FLUSHING VAVLE DB"."AGLV-301" AND NOT "P_TRIG".ARR[35];   // rising edge
   "P_TRIG".ARR[35] := "FLUSHING VAVLE DB"."AGLV-301";
   IF #_w1 THEN "HOOTER" := TRUE; END_IF;
END_REGION

REGION Network 37: RO-1 A AUTO FLUSING VALVE AGLV-301 CLOSE COMMOND FAIL
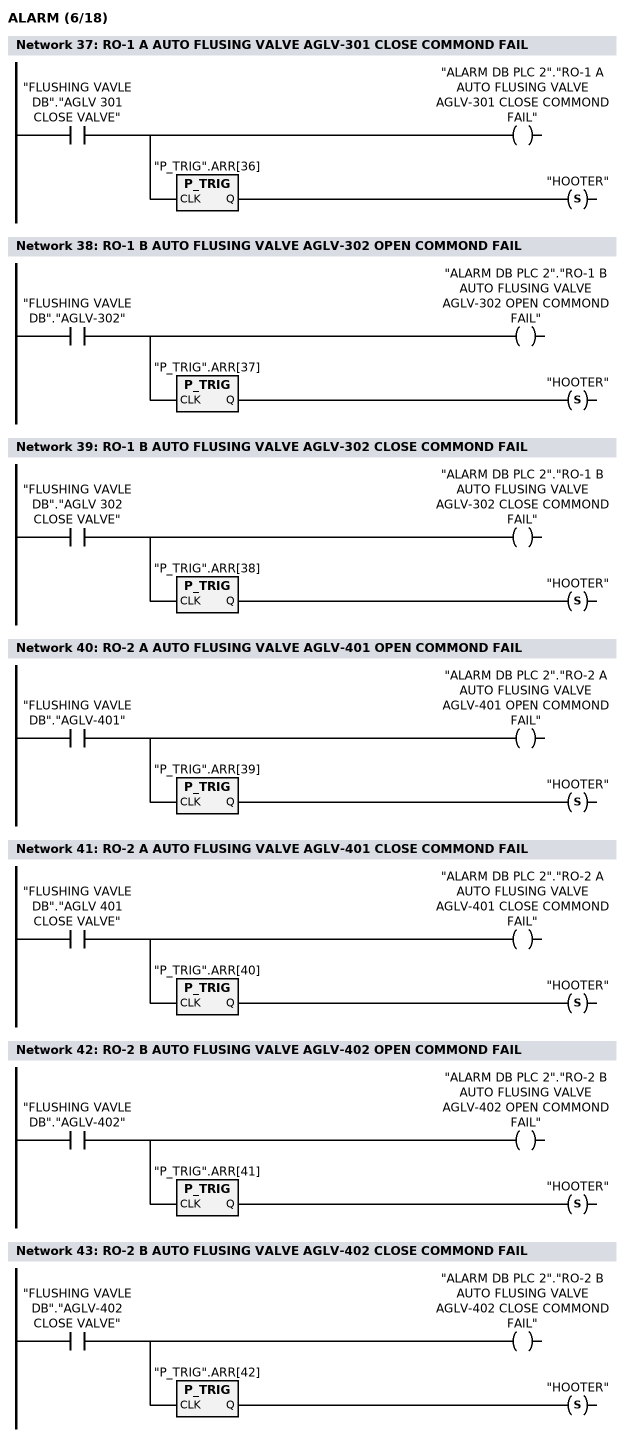
   RUNG wire#powerrail
      Contact( "FLUSHING VAVLE DB"."AGLV 301 CLOSE VALVE" )
      wire#w1
      Coil( "ALARM DB PLC 2"."RO-1 A AUTO FLUSING VALVE AGLV-301 CLOSE COMMOND FAIL" )
   END_RUNG
   RUNG wire#w1
      P_Trig( "P_TRIG".ARR[36] )
      S_Coil( "HOOTER" )
   END_RUNG
   // the same network as SCL:
   "ALARM DB PLC 2"."RO-1 A AUTO FLUSING VALVE AGLV-301 CLOSE COMMOND FAIL" := "FLUSHING VAVLE DB"."AGLV 301 CLOSE VALVE";
   #_w1 := "FLUSHING VAVLE DB"."AGLV 301 CLOSE VALVE" AND NOT "P_TRIG".ARR[36];   // rising edge
   "P_TRIG".ARR[36] := "FLUSHING VAVLE DB"."AGLV 301 CLOSE VALVE";
   IF #_w1 THEN "HOOTER" := TRUE; END_IF;
END_REGION

REGION Network 38: RO-1 B AUTO FLUSING VALVE AGLV-302 OPEN COMMOND FAIL
   RUNG wire#powerrail
      Contact( "FLUSHING VAVLE DB"."AGLV-302" )
      wire#w1
      Coil( "ALARM DB PLC 2"."RO-1 B AUTO FLUSING VALVE AGLV-302 OPEN COMMOND FAIL" )
   END_RUNG
   RUNG wire#w1
      P_Trig( "P_TRIG".ARR[37] )
      S_Coil( "HOOTER" )
   END_RUNG
   // the same network as SCL:
   "ALARM DB PLC 2"."RO-1 B AUTO FLUSING VALVE AGLV-302 OPEN COMMOND FAIL" := "FLUSHING VAVLE DB"."AGLV-302";
   #_w1 := "FLUSHING VAVLE DB"."AGLV-302" AND NOT "P_TRIG".ARR[37];   // rising edge
   "P_TRIG".ARR[37] := "FLUSHING VAVLE DB"."AGLV-302";
   IF #_w1 THEN "HOOTER" := TRUE; END_IF;
END_REGION

REGION Network 39: RO-1 B AUTO FLUSING VALVE AGLV-302 CLOSE COMMOND FAIL
   RUNG wire#powerrail
      Contact( "FLUSHING VAVLE DB"."AGLV 302 CLOSE VALVE" )
      wire#w1
      Coil( "ALARM DB PLC 2"."RO-1 B AUTO FLUSING VALVE AGLV-302 CLOSE COMMOND FAIL" )
   END_RUNG
   RUNG wire#w1
      P_Trig( "P_TRIG".ARR[38] )
      S_Coil( "HOOTER" )
   END_RUNG
   // the same network as SCL:
   "ALARM DB PLC 2"."RO-1 B AUTO FLUSING VALVE AGLV-302 CLOSE COMMOND FAIL" := "FLUSHING VAVLE DB"."AGLV 302 CLOSE VALVE";
   #_w1 := "FLUSHING VAVLE DB"."AGLV 302 CLOSE VALVE" AND NOT "P_TRIG".ARR[38];   // rising edge
   "P_TRIG".ARR[38] := "FLUSHING VAVLE DB"."AGLV 302 CLOSE VALVE";
   IF #_w1 THEN "HOOTER" := TRUE; END_IF;
END_REGION

REGION Network 40: RO-2 A AUTO FLUSING VALVE AGLV-401 OPEN COMMOND FAIL
   RUNG wire#powerrail
      Contact( "FLUSHING VAVLE DB"."AGLV-401" )
      wire#w1
      Coil( "ALARM DB PLC 2"."RO-2 A AUTO FLUSING VALVE AGLV-401 OPEN COMMOND FAIL" )
   END_RUNG
   RUNG wire#w1
      P_Trig( "P_TRIG".ARR[39] )
      S_Coil( "HOOTER" )
   END_RUNG
   // the same network as SCL:
   "ALARM DB PLC 2"."RO-2 A AUTO FLUSING VALVE AGLV-401 OPEN COMMOND FAIL" := "FLUSHING VAVLE DB"."AGLV-401";
   #_w1 := "FLUSHING VAVLE DB"."AGLV-401" AND NOT "P_TRIG".ARR[39];   // rising edge
   "P_TRIG".ARR[39] := "FLUSHING VAVLE DB"."AGLV-401";
   IF #_w1 THEN "HOOTER" := TRUE; END_IF;
END_REGION

REGION Network 41: RO-2 A AUTO FLUSING VALVE AGLV-401 CLOSE COMMOND FAIL
   RUNG wire#powerrail
      Contact( "FLUSHING VAVLE DB"."AGLV 401 CLOSE VALVE" )
      wire#w1
      Coil( "ALARM DB PLC 2"."RO-2 A AUTO FLUSING VALVE AGLV-401 CLOSE COMMOND FAIL" )
   END_RUNG
   RUNG wire#w1
      P_Trig( "P_TRIG".ARR[40] )
      S_Coil( "HOOTER" )
   END_RUNG
   // the same network as SCL:
   "ALARM DB PLC 2"."RO-2 A AUTO FLUSING VALVE AGLV-401 CLOSE COMMOND FAIL" := "FLUSHING VAVLE DB"."AGLV 401 CLOSE VALVE";
   #_w1 := "FLUSHING VAVLE DB"."AGLV 401 CLOSE VALVE" AND NOT "P_TRIG".ARR[40];   // rising edge
   "P_TRIG".ARR[40] := "FLUSHING VAVLE DB"."AGLV 401 CLOSE VALVE";
   IF #_w1 THEN "HOOTER" := TRUE; END_IF;
END_REGION

REGION Network 42: RO-2 B AUTO FLUSING VALVE AGLV-402 OPEN COMMOND FAIL
   RUNG wire#powerrail
      Contact( "FLUSHING VAVLE DB"."AGLV-402" )
      wire#w1
      Coil( "ALARM DB PLC 2"."RO-2 B AUTO FLUSING VALVE AGLV-402 OPEN COMMOND FAIL" )
   END_RUNG
   RUNG wire#w1
      P_Trig( "P_TRIG".ARR[41] )
      S_Coil( "HOOTER" )
   END_RUNG
   // the same network as SCL:
   "ALARM DB PLC 2"."RO-2 B AUTO FLUSING VALVE AGLV-402 OPEN COMMOND FAIL" := "FLUSHING VAVLE DB"."AGLV-402";
   #_w1 := "FLUSHING VAVLE DB"."AGLV-402" AND NOT "P_TRIG".ARR[41];   // rising edge
   "P_TRIG".ARR[41] := "FLUSHING VAVLE DB"."AGLV-402";
   IF #_w1 THEN "HOOTER" := TRUE; END_IF;
END_REGION

REGION Network 43: RO-2 B AUTO FLUSING VALVE AGLV-402 CLOSE COMMOND FAIL
   RUNG wire#powerrail
      Contact( "FLUSHING VAVLE DB"."AGLV-402 CLOSE VALVE" )
      wire#w1
      Coil( "ALARM DB PLC 2"."RO-2 B AUTO FLUSING VALVE AGLV-402 CLOSE COMMOND FAIL" )
   END_RUNG
   RUNG wire#w1
      P_Trig( "P_TRIG".ARR[42] )
      S_Coil( "HOOTER" )
   END_RUNG
   // the same network as SCL:
   "ALARM DB PLC 2"."RO-2 B AUTO FLUSING VALVE AGLV-402 CLOSE COMMOND FAIL" := "FLUSHING VAVLE DB"."AGLV-402 CLOSE VALVE";
   #_w1 := "FLUSHING VAVLE DB"."AGLV-402 CLOSE VALVE" AND NOT "P_TRIG".ARR[42];   // rising edge
   "P_TRIG".ARR[42] := "FLUSHING VAVLE DB"."AGLV-402 CLOSE VALVE";
   IF #_w1 THEN "HOOTER" := TRUE; END_IF;
END_REGION

REGION Network 44: EDI AUTO DUMP VALVE ABV-501 OPEN COMMOND FAIL
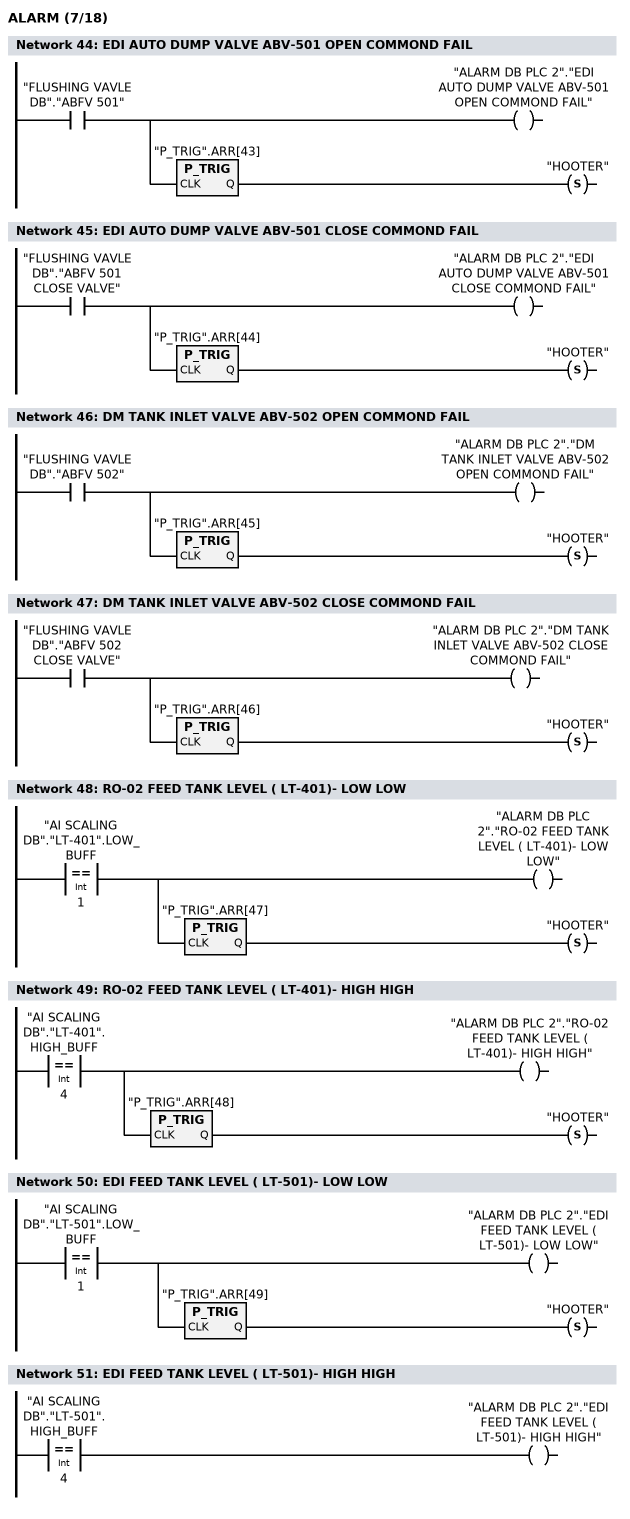
   RUNG wire#powerrail
      Contact( "FLUSHING VAVLE DB"."ABFV 501" )
      wire#w1
      Coil( "ALARM DB PLC 2"."EDI AUTO DUMP VALVE ABV-501 OPEN COMMOND FAIL" )
   END_RUNG
   RUNG wire#w1
      P_Trig( "P_TRIG".ARR[43] )
      S_Coil( "HOOTER" )
   END_RUNG
   // the same network as SCL:
   "ALARM DB PLC 2"."EDI AUTO DUMP VALVE ABV-501 OPEN COMMOND FAIL" := "FLUSHING VAVLE DB"."ABFV 501";
   #_w1 := "FLUSHING VAVLE DB"."ABFV 501" AND NOT "P_TRIG".ARR[43];   // rising edge
   "P_TRIG".ARR[43] := "FLUSHING VAVLE DB"."ABFV 501";
   IF #_w1 THEN "HOOTER" := TRUE; END_IF;
END_REGION

REGION Network 45: EDI AUTO DUMP VALVE ABV-501 CLOSE COMMOND FAIL
   RUNG wire#powerrail
      Contact( "FLUSHING VAVLE DB"."ABFV 501 CLOSE VALVE" )
      wire#w1
      Coil( "ALARM DB PLC 2"."EDI AUTO DUMP VALVE ABV-501 CLOSE COMMOND FAIL" )
   END_RUNG
   RUNG wire#w1
      P_Trig( "P_TRIG".ARR[44] )
      S_Coil( "HOOTER" )
   END_RUNG
   // the same network as SCL:
   "ALARM DB PLC 2"."EDI AUTO DUMP VALVE ABV-501 CLOSE COMMOND FAIL" := "FLUSHING VAVLE DB"."ABFV 501 CLOSE VALVE";
   #_w1 := "FLUSHING VAVLE DB"."ABFV 501 CLOSE VALVE" AND NOT "P_TRIG".ARR[44];   // rising edge
   "P_TRIG".ARR[44] := "FLUSHING VAVLE DB"."ABFV 501 CLOSE VALVE";
   IF #_w1 THEN "HOOTER" := TRUE; END_IF;
END_REGION

REGION Network 46: DM TANK INLET VALVE ABV-502 OPEN COMMOND FAIL
   RUNG wire#powerrail
      Contact( "FLUSHING VAVLE DB"."ABFV 502" )
      wire#w1
      Coil( "ALARM DB PLC 2"."DM TANK INLET VALVE ABV-502 OPEN COMMOND FAIL" )
   END_RUNG
   RUNG wire#w1
      P_Trig( "P_TRIG".ARR[45] )
      S_Coil( "HOOTER" )
   END_RUNG
   // the same network as SCL:
   "ALARM DB PLC 2"."DM TANK INLET VALVE ABV-502 OPEN COMMOND FAIL" := "FLUSHING VAVLE DB"."ABFV 502";
   #_w1 := "FLUSHING VAVLE DB"."ABFV 502" AND NOT "P_TRIG".ARR[45];   // rising edge
   "P_TRIG".ARR[45] := "FLUSHING VAVLE DB"."ABFV 502";
   IF #_w1 THEN "HOOTER" := TRUE; END_IF;
END_REGION

REGION Network 47: DM TANK INLET VALVE ABV-502 CLOSE COMMOND FAIL
   RUNG wire#powerrail
      Contact( "FLUSHING VAVLE DB"."ABFV 502 CLOSE VALVE" )
      wire#w1
      Coil( "ALARM DB PLC 2"."DM TANK INLET VALVE ABV-502 CLOSE COMMOND FAIL" )
   END_RUNG
   RUNG wire#w1
      P_Trig( "P_TRIG".ARR[46] )
      S_Coil( "HOOTER" )
   END_RUNG
   // the same network as SCL:
   "ALARM DB PLC 2"."DM TANK INLET VALVE ABV-502 CLOSE COMMOND FAIL" := "FLUSHING VAVLE DB"."ABFV 502 CLOSE VALVE";
   #_w1 := "FLUSHING VAVLE DB"."ABFV 502 CLOSE VALVE" AND NOT "P_TRIG".ARR[46];   // rising edge
   "P_TRIG".ARR[46] := "FLUSHING VAVLE DB"."ABFV 502 CLOSE VALVE";
   IF #_w1 THEN "HOOTER" := TRUE; END_IF;
END_REGION

REGION Network 48: RO-02 FEED TANK LEVEL ( LT-401)- LOW LOW
   RUNG wire#powerrail
      { S7_Templates := "SrcType := Int" } EQ_Contact(in1 := "AI SCALING DB"."LT-401".LOW_BUFF, in2 := 1)
      wire#w1
      Coil( "ALARM DB PLC 2"."RO-02 FEED TANK LEVEL ( LT-401)- LOW LOW" )
   END_RUNG
   RUNG wire#w1
      P_Trig( "P_TRIG".ARR[47] )
      S_Coil( "HOOTER" )
   END_RUNG
   // the same network as SCL:
   "ALARM DB PLC 2"."RO-02 FEED TANK LEVEL ( LT-401)- LOW LOW" := "AI SCALING DB"."LT-401".LOW_BUFF = 1;
   #_w1 := "ALARM DB PLC 2"."RO-02 FEED TANK LEVEL ( LT-401)- LOW LOW" AND NOT "P_TRIG".ARR[47];   // rising edge
   "P_TRIG".ARR[47] := "ALARM DB PLC 2"."RO-02 FEED TANK LEVEL ( LT-401)- LOW LOW";
   IF #_w1 THEN "HOOTER" := TRUE; END_IF;
END_REGION

REGION Network 49: RO-02 FEED TANK LEVEL ( LT-401)- HIGH HIGH
   RUNG wire#powerrail
      { S7_Templates := "SrcType := Int" } EQ_Contact(in1 := "AI SCALING DB"."LT-401".HIGH_BUFF, in2 := 4)
      wire#w1
      Coil( "ALARM DB PLC 2"."RO-02 FEED TANK LEVEL ( LT-401)- HIGH HIGH" )
   END_RUNG
   RUNG wire#w1
      P_Trig( "P_TRIG".ARR[48] )
      S_Coil( "HOOTER" )
   END_RUNG
   // the same network as SCL:
   "ALARM DB PLC 2"."RO-02 FEED TANK LEVEL ( LT-401)- HIGH HIGH" := "AI SCALING DB"."LT-401".HIGH_BUFF = 4;
   #_w1 := "ALARM DB PLC 2"."RO-02 FEED TANK LEVEL ( LT-401)- HIGH HIGH" AND NOT "P_TRIG".ARR[48];   // rising edge
   "P_TRIG".ARR[48] := "ALARM DB PLC 2"."RO-02 FEED TANK LEVEL ( LT-401)- HIGH HIGH";
   IF #_w1 THEN "HOOTER" := TRUE; END_IF;
END_REGION

REGION Network 50: EDI FEED TANK LEVEL ( LT-501)- LOW LOW
   RUNG wire#powerrail
      { S7_Templates := "SrcType := Int" } EQ_Contact(in1 := "AI SCALING DB"."LT-501".LOW_BUFF, in2 := 1)
      wire#w1
      Coil( "ALARM DB PLC 2"."EDI FEED TANK LEVEL ( LT-501)- LOW LOW" )
   END_RUNG
   RUNG wire#w1
      P_Trig( "P_TRIG".ARR[49] )
      S_Coil( "HOOTER" )
   END_RUNG
   // the same network as SCL:
   "ALARM DB PLC 2"."EDI FEED TANK LEVEL ( LT-501)- LOW LOW" := "AI SCALING DB"."LT-501".LOW_BUFF = 1;
   #_w1 := "ALARM DB PLC 2"."EDI FEED TANK LEVEL ( LT-501)- LOW LOW" AND NOT "P_TRIG".ARR[49];   // rising edge
   "P_TRIG".ARR[49] := "ALARM DB PLC 2"."EDI FEED TANK LEVEL ( LT-501)- LOW LOW";
   IF #_w1 THEN "HOOTER" := TRUE; END_IF;
END_REGION

REGION Network 51: EDI FEED TANK LEVEL ( LT-501)- HIGH HIGH
   RUNG wire#powerrail
      { S7_Templates := "SrcType := Int" } EQ_Contact(in1 := "AI SCALING DB"."LT-501".HIGH_BUFF, in2 := 4)
      Coil( "ALARM DB PLC 2"."EDI FEED TANK LEVEL ( LT-501)- HIGH HIGH" )
   END_RUNG
   // the same network as SCL:
   "ALARM DB PLC 2"."EDI FEED TANK LEVEL ( LT-501)- HIGH HIGH" := "AI SCALING DB"."LT-501".HIGH_BUFF = 4;
END_REGION

REGION Network 52: DM WATER STORAGE TANK LEVEL ( LT-502)- LOW LOW
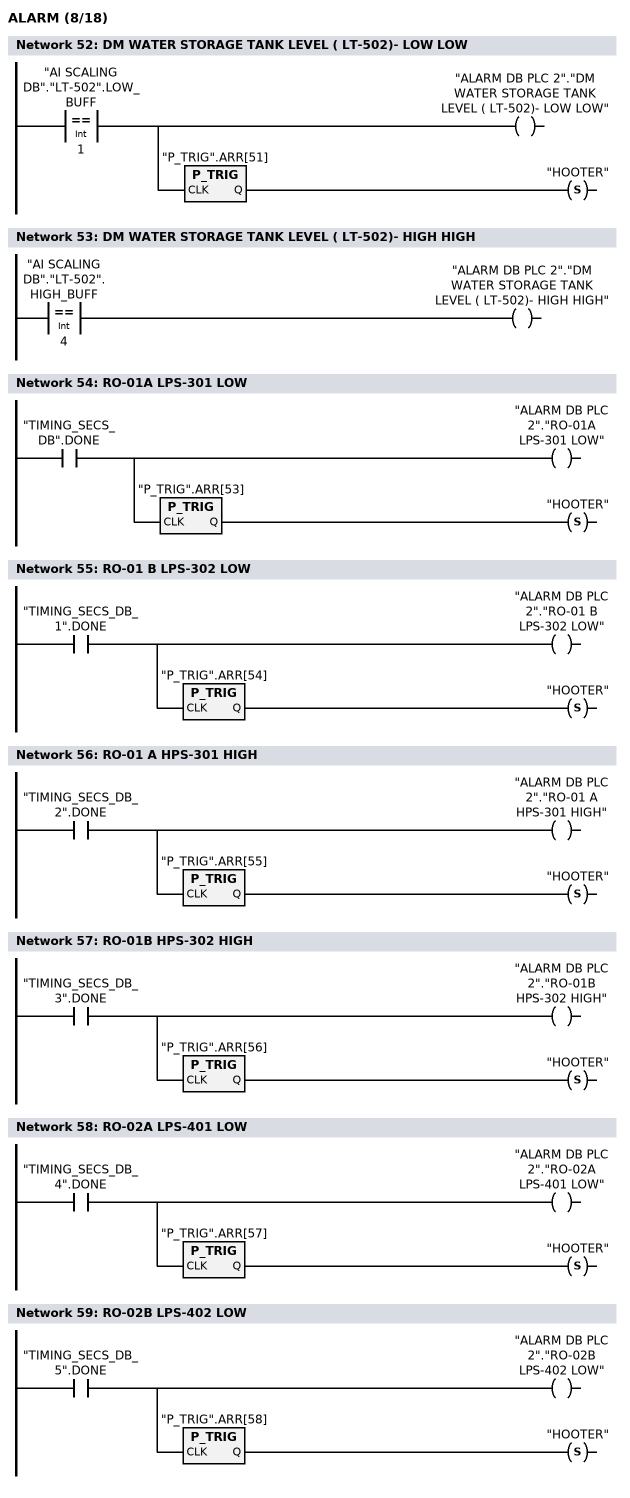
   RUNG wire#powerrail
      { S7_Templates := "SrcType := Int" } EQ_Contact(in1 := "AI SCALING DB"."LT-502".LOW_BUFF, in2 := 1)
      wire#w1
      Coil( "ALARM DB PLC 2"."DM WATER STORAGE TANK  LEVEL ( LT-502)- LOW LOW" )
   END_RUNG
   RUNG wire#w1
      P_Trig( "P_TRIG".ARR[51] )
      S_Coil( "HOOTER" )
   END_RUNG
   // the same network as SCL:
   "ALARM DB PLC 2"."DM WATER STORAGE TANK  LEVEL ( LT-502)- LOW LOW" := "AI SCALING DB"."LT-502".LOW_BUFF = 1;
   #_w1 := "ALARM DB PLC 2"."DM WATER STORAGE TANK  LEVEL ( LT-502)- LOW LOW" AND NOT "P_TRIG".ARR[51];   // rising edge
   "P_TRIG".ARR[51] := "ALARM DB PLC 2"."DM WATER STORAGE TANK  LEVEL ( LT-502)- LOW LOW";
   IF #_w1 THEN "HOOTER" := TRUE; END_IF;
END_REGION

REGION Network 53: DM WATER STORAGE TANK LEVEL ( LT-502)- HIGH HIGH
   RUNG wire#powerrail
      { S7_Templates := "SrcType := Int" } EQ_Contact(in1 := "AI SCALING DB"."LT-502".HIGH_BUFF, in2 := 4)
      Coil( "ALARM DB PLC 2"."DM WATER STORAGE TANK LEVEL ( LT-502)- HIGH HIGH" )
   END_RUNG
   // the same network as SCL:
   "ALARM DB PLC 2"."DM WATER STORAGE TANK LEVEL ( LT-502)- HIGH HIGH" := "AI SCALING DB"."LT-502".HIGH_BUFF = 4;
END_REGION

REGION Network 54: RO-01A LPS-301 LOW
   RUNG wire#powerrail
      Contact( "TIMING_SECS_DB".DONE )
      wire#w1
      Coil( "ALARM DB PLC 2"."RO-01A LPS-301 LOW" )
   END_RUNG
   RUNG wire#w1
      P_Trig( "P_TRIG".ARR[53] )
      S_Coil( "HOOTER" )
   END_RUNG
   // the same network as SCL:
   "ALARM DB PLC 2"."RO-01A LPS-301 LOW" := "TIMING_SECS_DB".DONE;
   #_w1 := "TIMING_SECS_DB".DONE AND NOT "P_TRIG".ARR[53];   // rising edge
   "P_TRIG".ARR[53] := "TIMING_SECS_DB".DONE;
   IF #_w1 THEN "HOOTER" := TRUE; END_IF;
END_REGION

REGION Network 55: RO-01 B LPS-302 LOW
   RUNG wire#powerrail
      Contact( "TIMING_SECS_DB_1".DONE )
      wire#w1
      Coil( "ALARM DB PLC 2"."RO-01 B LPS-302 LOW" )
   END_RUNG
   RUNG wire#w1
      P_Trig( "P_TRIG".ARR[54] )
      S_Coil( "HOOTER" )
   END_RUNG
   // the same network as SCL:
   "ALARM DB PLC 2"."RO-01 B LPS-302 LOW" := "TIMING_SECS_DB_1".DONE;
   #_w1 := "TIMING_SECS_DB_1".DONE AND NOT "P_TRIG".ARR[54];   // rising edge
   "P_TRIG".ARR[54] := "TIMING_SECS_DB_1".DONE;
   IF #_w1 THEN "HOOTER" := TRUE; END_IF;
END_REGION

REGION Network 56: RO-01 A HPS-301 HIGH
   RUNG wire#powerrail
      Contact( "TIMING_SECS_DB_2".DONE )
      wire#w1
      Coil( "ALARM DB PLC 2"."RO-01 A HPS-301 HIGH" )
   END_RUNG
   RUNG wire#w1
      P_Trig( "P_TRIG".ARR[55] )
      S_Coil( "HOOTER" )
   END_RUNG
   // the same network as SCL:
   "ALARM DB PLC 2"."RO-01 A HPS-301 HIGH" := "TIMING_SECS_DB_2".DONE;
   #_w1 := "TIMING_SECS_DB_2".DONE AND NOT "P_TRIG".ARR[55];   // rising edge
   "P_TRIG".ARR[55] := "TIMING_SECS_DB_2".DONE;
   IF #_w1 THEN "HOOTER" := TRUE; END_IF;
END_REGION

REGION Network 57: RO-01B HPS-302 HIGH
   RUNG wire#powerrail
      Contact( "TIMING_SECS_DB_3".DONE )
      wire#w1
      Coil( "ALARM DB PLC 2"."RO-01B HPS-302 HIGH" )
   END_RUNG
   RUNG wire#w1
      P_Trig( "P_TRIG".ARR[56] )
      S_Coil( "HOOTER" )
   END_RUNG
   // the same network as SCL:
   "ALARM DB PLC 2"."RO-01B HPS-302 HIGH" := "TIMING_SECS_DB_3".DONE;
   #_w1 := "TIMING_SECS_DB_3".DONE AND NOT "P_TRIG".ARR[56];   // rising edge
   "P_TRIG".ARR[56] := "TIMING_SECS_DB_3".DONE;
   IF #_w1 THEN "HOOTER" := TRUE; END_IF;
END_REGION

REGION Network 58: RO-02A LPS-401 LOW
   RUNG wire#powerrail
      Contact( "TIMING_SECS_DB_4".DONE )
      wire#w1
      Coil( "ALARM DB PLC 2"."RO-02A LPS-401 LOW" )
   END_RUNG
   RUNG wire#w1
      P_Trig( "P_TRIG".ARR[57] )
      S_Coil( "HOOTER" )
   END_RUNG
   // the same network as SCL:
   "ALARM DB PLC 2"."RO-02A LPS-401 LOW" := "TIMING_SECS_DB_4".DONE;
   #_w1 := "TIMING_SECS_DB_4".DONE AND NOT "P_TRIG".ARR[57];   // rising edge
   "P_TRIG".ARR[57] := "TIMING_SECS_DB_4".DONE;
   IF #_w1 THEN "HOOTER" := TRUE; END_IF;
END_REGION

REGION Network 59: RO-02B LPS-402 LOW
   RUNG wire#powerrail
      Contact( "TIMING_SECS_DB_5".DONE )
      wire#w1
      Coil( "ALARM DB PLC 2"."RO-02B LPS-402 LOW" )
   END_RUNG
   RUNG wire#w1
      P_Trig( "P_TRIG".ARR[58] )
      S_Coil( "HOOTER" )
   END_RUNG
   // the same network as SCL:
   "ALARM DB PLC 2"."RO-02B LPS-402 LOW" := "TIMING_SECS_DB_5".DONE;
   #_w1 := "TIMING_SECS_DB_5".DONE AND NOT "P_TRIG".ARR[58];   // rising edge
   "P_TRIG".ARR[58] := "TIMING_SECS_DB_5".DONE;
   IF #_w1 THEN "HOOTER" := TRUE; END_IF;
END_REGION

REGION Network 60: RO-02A HPS-401 HIGH
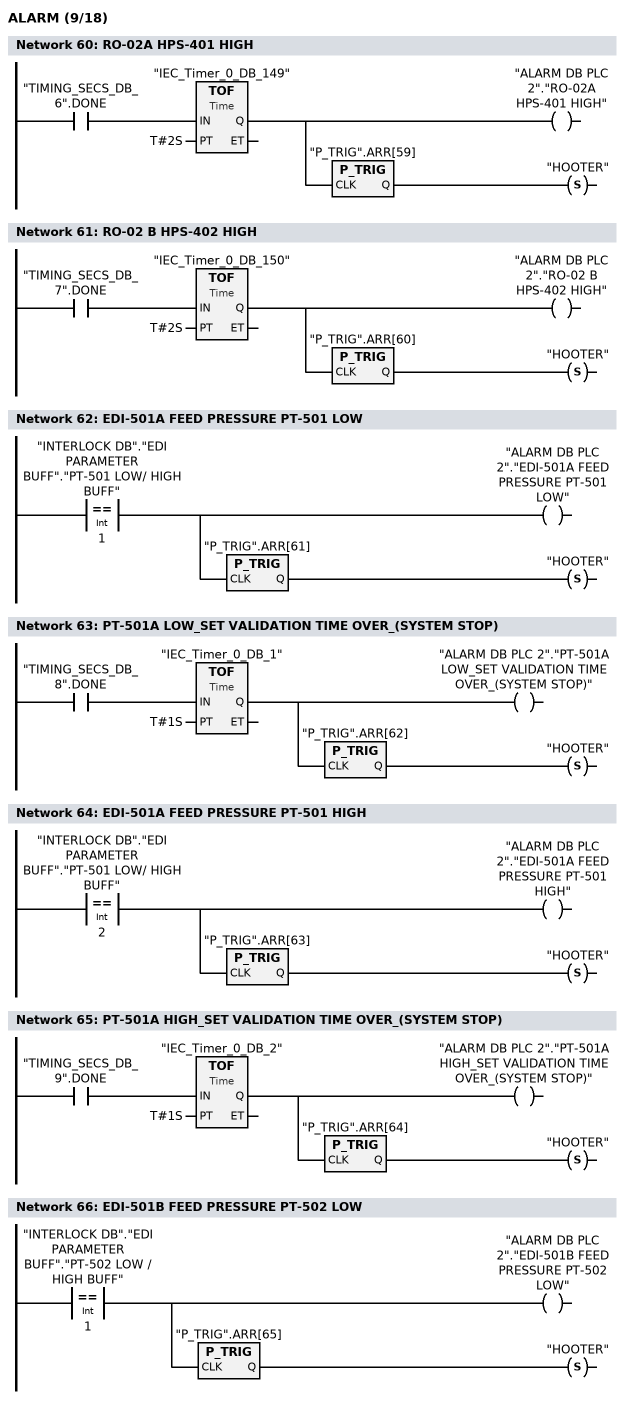
   RUNG wire#powerrail
      Contact( "TIMING_SECS_DB_6".DONE )
      { S7_Templates := "time_type := Time" } "IEC_Timer_0_DB_149".TOF(pt := T#2S, et =>)
      wire#w1
      Coil( "ALARM DB PLC 2"."RO-02A HPS-401 HIGH" )
   END_RUNG
   RUNG wire#w1
      P_Trig( "P_TRIG".ARR[59] )
      S_Coil( "HOOTER" )
   END_RUNG
   // the same network as SCL:
   "IEC_Timer_0_DB_149".TOF(IN := "TIMING_SECS_DB_6".DONE, PT := T#2S);
   "ALARM DB PLC 2"."RO-02A HPS-401 HIGH" := "IEC_Timer_0_DB_149".Q;
   #_w1 := "IEC_Timer_0_DB_149".Q AND NOT "P_TRIG".ARR[59];   // rising edge
   "P_TRIG".ARR[59] := "IEC_Timer_0_DB_149".Q;
   IF #_w1 THEN "HOOTER" := TRUE; END_IF;
END_REGION

REGION Network 61: RO-02 B HPS-402 HIGH
   RUNG wire#powerrail
      Contact( "TIMING_SECS_DB_7".DONE )
      { S7_Templates := "time_type := Time" } "IEC_Timer_0_DB_150".TOF(pt := T#2S, et =>)
      wire#w1
      Coil( "ALARM DB PLC 2"."RO-02 B HPS-402 HIGH" )
   END_RUNG
   RUNG wire#w1
      P_Trig( "P_TRIG".ARR[60] )
      S_Coil( "HOOTER" )
   END_RUNG
   // the same network as SCL:
   "IEC_Timer_0_DB_150".TOF(IN := "TIMING_SECS_DB_7".DONE, PT := T#2S);
   "ALARM DB PLC 2"."RO-02 B HPS-402 HIGH" := "IEC_Timer_0_DB_150".Q;
   #_w1 := "IEC_Timer_0_DB_150".Q AND NOT "P_TRIG".ARR[60];   // rising edge
   "P_TRIG".ARR[60] := "IEC_Timer_0_DB_150".Q;
   IF #_w1 THEN "HOOTER" := TRUE; END_IF;
END_REGION

REGION Network 62: EDI-501A FEED PRESSURE PT-501 LOW
   RUNG wire#powerrail
      { S7_Templates := "SrcType := Int" } EQ_Contact(in1 := "INTERLOCK DB"."EDI PARAMETER BUFF"."PT-501 LOW/ HIGH BUFF", in2 := 1)
      wire#w1
      Coil( "ALARM DB PLC 2"."EDI-501A FEED PRESSURE PT-501 LOW" )
   END_RUNG
   RUNG wire#w1
      P_Trig( "P_TRIG".ARR[61] )
      S_Coil( "HOOTER" )
   END_RUNG
   // the same network as SCL:
   "ALARM DB PLC 2"."EDI-501A FEED PRESSURE PT-501 LOW" := "INTERLOCK DB"."EDI PARAMETER BUFF"."PT-501 LOW/ HIGH BUFF" = 1;
   #_w1 := "ALARM DB PLC 2"."EDI-501A FEED PRESSURE PT-501 LOW" AND NOT "P_TRIG".ARR[61];   // rising edge
   "P_TRIG".ARR[61] := "ALARM DB PLC 2"."EDI-501A FEED PRESSURE PT-501 LOW";
   IF #_w1 THEN "HOOTER" := TRUE; END_IF;
END_REGION

REGION Network 63: PT-501A LOW_SET VALIDATION TIME OVER_(SYSTEM STOP)
   RUNG wire#powerrail
      Contact( "TIMING_SECS_DB_8".DONE )
      { S7_Templates := "time_type := Time" } "IEC_Timer_0_DB_1".TOF(pt := T#1S, et =>)
      wire#w1
      Coil( "ALARM DB PLC 2"."PT-501A LOW_SET VALIDATION TIME OVER_(SYSTEM STOP)" )
   END_RUNG
   RUNG wire#w1
      P_Trig( "P_TRIG".ARR[62] )
      S_Coil( "HOOTER" )
   END_RUNG
   // the same network as SCL:
   "IEC_Timer_0_DB_1".TOF(IN := "TIMING_SECS_DB_8".DONE, PT := T#1S);
   "ALARM DB PLC 2"."PT-501A LOW_SET VALIDATION TIME OVER_(SYSTEM STOP)" := "IEC_Timer_0_DB_1".Q;
   #_w1 := "IEC_Timer_0_DB_1".Q AND NOT "P_TRIG".ARR[62];   // rising edge
   "P_TRIG".ARR[62] := "IEC_Timer_0_DB_1".Q;
   IF #_w1 THEN "HOOTER" := TRUE; END_IF;
END_REGION

REGION Network 64: EDI-501A FEED PRESSURE PT-501 HIGH
   RUNG wire#powerrail
      { S7_Templates := "SrcType := Int" } EQ_Contact(in1 := "INTERLOCK DB"."EDI PARAMETER BUFF"."PT-501 LOW/ HIGH BUFF", in2 := 2)
      wire#w1
      Coil( "ALARM DB PLC 2"."EDI-501A FEED PRESSURE PT-501 HIGH" )
   END_RUNG
   RUNG wire#w1
      P_Trig( "P_TRIG".ARR[63] )
      S_Coil( "HOOTER" )
   END_RUNG
   // the same network as SCL:
   "ALARM DB PLC 2"."EDI-501A FEED PRESSURE PT-501 HIGH" := "INTERLOCK DB"."EDI PARAMETER BUFF"."PT-501 LOW/ HIGH BUFF" = 2;
   #_w1 := "ALARM DB PLC 2"."EDI-501A FEED PRESSURE PT-501 HIGH" AND NOT "P_TRIG".ARR[63];   // rising edge
   "P_TRIG".ARR[63] := "ALARM DB PLC 2"."EDI-501A FEED PRESSURE PT-501 HIGH";
   IF #_w1 THEN "HOOTER" := TRUE; END_IF;
END_REGION

REGION Network 65: PT-501A HIGH_SET VALIDATION TIME OVER_(SYSTEM STOP)
   RUNG wire#powerrail
      Contact( "TIMING_SECS_DB_9".DONE )
      { S7_Templates := "time_type := Time" } "IEC_Timer_0_DB_2".TOF(pt := T#1S, et =>)
      wire#w1
      Coil( "ALARM DB PLC 2"."PT-501A HIGH_SET VALIDATION TIME OVER_(SYSTEM STOP)" )
   END_RUNG
   RUNG wire#w1
      P_Trig( "P_TRIG".ARR[64] )
      S_Coil( "HOOTER" )
   END_RUNG
   // the same network as SCL:
   "IEC_Timer_0_DB_2".TOF(IN := "TIMING_SECS_DB_9".DONE, PT := T#1S);
   "ALARM DB PLC 2"."PT-501A HIGH_SET VALIDATION TIME OVER_(SYSTEM STOP)" := "IEC_Timer_0_DB_2".Q;
   #_w1 := "IEC_Timer_0_DB_2".Q AND NOT "P_TRIG".ARR[64];   // rising edge
   "P_TRIG".ARR[64] := "IEC_Timer_0_DB_2".Q;
   IF #_w1 THEN "HOOTER" := TRUE; END_IF;
END_REGION

REGION Network 66: EDI-501B FEED PRESSURE PT-502 LOW
   RUNG wire#powerrail
      { S7_Templates := "SrcType := Int" } EQ_Contact(in1 := "INTERLOCK DB"."EDI PARAMETER BUFF"."PT-502 LOW / HIGH BUFF", in2 := 1)
      wire#w1
      Coil( "ALARM DB PLC 2"."EDI-501B FEED PRESSURE PT-502 LOW" )
   END_RUNG
   RUNG wire#w1
      P_Trig( "P_TRIG".ARR[65] )
      S_Coil( "HOOTER" )
   END_RUNG
   // the same network as SCL:
   "ALARM DB PLC 2"."EDI-501B FEED PRESSURE PT-502 LOW" := "INTERLOCK DB"."EDI PARAMETER BUFF"."PT-502 LOW / HIGH BUFF" = 1;
   #_w1 := "ALARM DB PLC 2"."EDI-501B FEED PRESSURE PT-502 LOW" AND NOT "P_TRIG".ARR[65];   // rising edge
   "P_TRIG".ARR[65] := "ALARM DB PLC 2"."EDI-501B FEED PRESSURE PT-502 LOW";
   IF #_w1 THEN "HOOTER" := TRUE; END_IF;
END_REGION

REGION Network 67: PT-501B LOW_SET VALIDATION TIME OVER_(SYSTEM STOP)
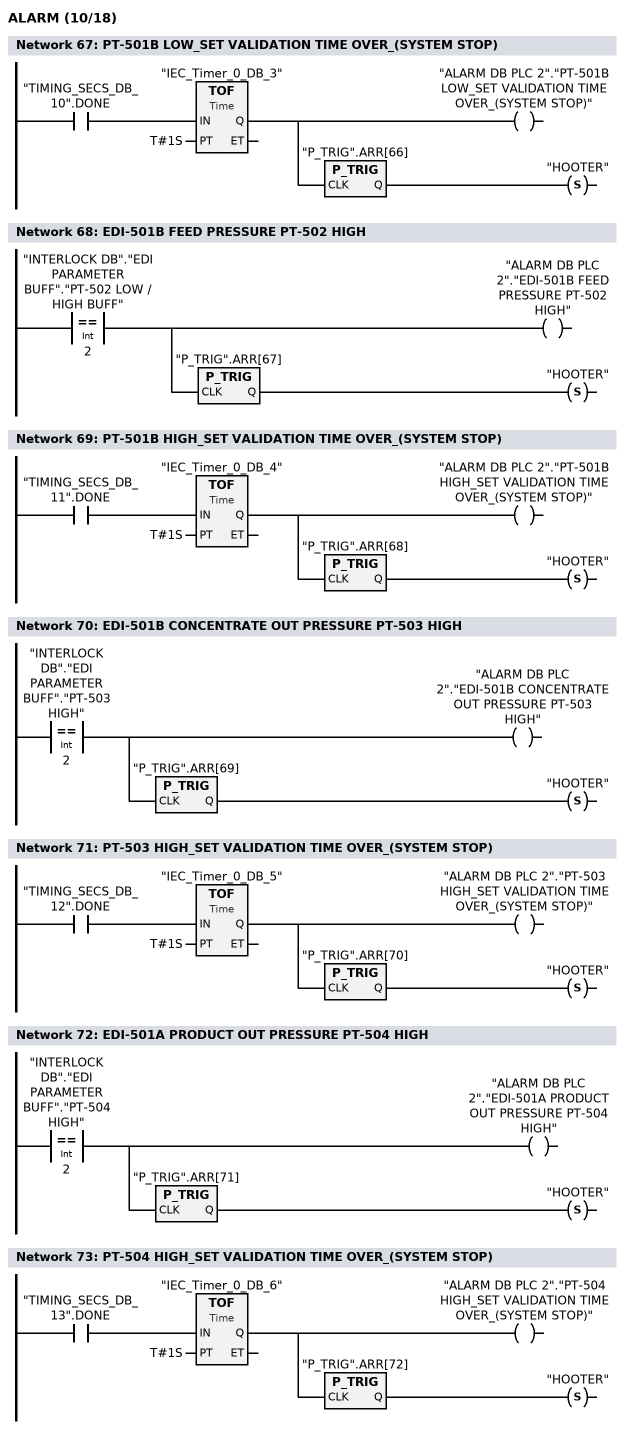
   RUNG wire#powerrail
      Contact( "TIMING_SECS_DB_10".DONE )
      { S7_Templates := "time_type := Time" } "IEC_Timer_0_DB_3".TOF(pt := T#1S, et =>)
      wire#w1
      Coil( "ALARM DB PLC 2"."PT-501B LOW_SET VALIDATION TIME OVER_(SYSTEM STOP)" )
   END_RUNG
   RUNG wire#w1
      P_Trig( "P_TRIG".ARR[66] )
      S_Coil( "HOOTER" )
   END_RUNG
   // the same network as SCL:
   "IEC_Timer_0_DB_3".TOF(IN := "TIMING_SECS_DB_10".DONE, PT := T#1S);
   "ALARM DB PLC 2"."PT-501B LOW_SET VALIDATION TIME OVER_(SYSTEM STOP)" := "IEC_Timer_0_DB_3".Q;
   #_w1 := "IEC_Timer_0_DB_3".Q AND NOT "P_TRIG".ARR[66];   // rising edge
   "P_TRIG".ARR[66] := "IEC_Timer_0_DB_3".Q;
   IF #_w1 THEN "HOOTER" := TRUE; END_IF;
END_REGION

REGION Network 68: EDI-501B FEED PRESSURE PT-502 HIGH
   RUNG wire#powerrail
      { S7_Templates := "SrcType := Int" } EQ_Contact(in1 := "INTERLOCK DB"."EDI PARAMETER BUFF"."PT-502 LOW / HIGH BUFF", in2 := 2)
      wire#w1
      Coil( "ALARM DB PLC 2"."EDI-501B FEED PRESSURE PT-502 HIGH" )
   END_RUNG
   RUNG wire#w1
      P_Trig( "P_TRIG".ARR[67] )
      S_Coil( "HOOTER" )
   END_RUNG
   // the same network as SCL:
   "ALARM DB PLC 2"."EDI-501B FEED PRESSURE PT-502 HIGH" := "INTERLOCK DB"."EDI PARAMETER BUFF"."PT-502 LOW / HIGH BUFF" = 2;
   #_w1 := "ALARM DB PLC 2"."EDI-501B FEED PRESSURE PT-502 HIGH" AND NOT "P_TRIG".ARR[67];   // rising edge
   "P_TRIG".ARR[67] := "ALARM DB PLC 2"."EDI-501B FEED PRESSURE PT-502 HIGH";
   IF #_w1 THEN "HOOTER" := TRUE; END_IF;
END_REGION

REGION Network 69: PT-501B HIGH_SET VALIDATION TIME OVER_(SYSTEM STOP)
   RUNG wire#powerrail
      Contact( "TIMING_SECS_DB_11".DONE )
      { S7_Templates := "time_type := Time" } "IEC_Timer_0_DB_4".TOF(pt := T#1S, et =>)
      wire#w1
      Coil( "ALARM DB PLC 2"."PT-501B HIGH_SET VALIDATION TIME OVER_(SYSTEM STOP)" )
   END_RUNG
   RUNG wire#w1
      P_Trig( "P_TRIG".ARR[68] )
      S_Coil( "HOOTER" )
   END_RUNG
   // the same network as SCL:
   "IEC_Timer_0_DB_4".TOF(IN := "TIMING_SECS_DB_11".DONE, PT := T#1S);
   "ALARM DB PLC 2"."PT-501B HIGH_SET VALIDATION TIME OVER_(SYSTEM STOP)" := "IEC_Timer_0_DB_4".Q;
   #_w1 := "IEC_Timer_0_DB_4".Q AND NOT "P_TRIG".ARR[68];   // rising edge
   "P_TRIG".ARR[68] := "IEC_Timer_0_DB_4".Q;
   IF #_w1 THEN "HOOTER" := TRUE; END_IF;
END_REGION

REGION Network 70: EDI-501B CONCENTRATE OUT PRESSURE PT-503 HIGH
   RUNG wire#powerrail
      { S7_Templates := "SrcType := Int" } EQ_Contact(in1 := "INTERLOCK DB"."EDI PARAMETER BUFF"."PT-503 HIGH", in2 := 2)
      wire#w1
      Coil( "ALARM DB PLC 2"."EDI-501B CONCENTRATE OUT PRESSURE PT-503 HIGH" )
   END_RUNG
   RUNG wire#w1
      P_Trig( "P_TRIG".ARR[69] )
      S_Coil( "HOOTER" )
   END_RUNG
   // the same network as SCL:
   "ALARM DB PLC 2"."EDI-501B CONCENTRATE OUT PRESSURE PT-503 HIGH" := "INTERLOCK DB"."EDI PARAMETER BUFF"."PT-503 HIGH" = 2;
   #_w1 := "ALARM DB PLC 2"."EDI-501B CONCENTRATE OUT PRESSURE PT-503 HIGH" AND NOT "P_TRIG".ARR[69];   // rising edge
   "P_TRIG".ARR[69] := "ALARM DB PLC 2"."EDI-501B CONCENTRATE OUT PRESSURE PT-503 HIGH";
   IF #_w1 THEN "HOOTER" := TRUE; END_IF;
END_REGION

REGION Network 71: PT-503 HIGH_SET VALIDATION TIME OVER_(SYSTEM STOP)
   RUNG wire#powerrail
      Contact( "TIMING_SECS_DB_12".DONE )
      { S7_Templates := "time_type := Time" } "IEC_Timer_0_DB_5".TOF(pt := T#1S, et =>)
      wire#w1
      Coil( "ALARM DB PLC 2"."PT-503 HIGH_SET VALIDATION TIME OVER_(SYSTEM STOP)" )
   END_RUNG
   RUNG wire#w1
      P_Trig( "P_TRIG".ARR[70] )
      S_Coil( "HOOTER" )
   END_RUNG
   // the same network as SCL:
   "IEC_Timer_0_DB_5".TOF(IN := "TIMING_SECS_DB_12".DONE, PT := T#1S);
   "ALARM DB PLC 2"."PT-503 HIGH_SET VALIDATION TIME OVER_(SYSTEM STOP)" := "IEC_Timer_0_DB_5".Q;
   #_w1 := "IEC_Timer_0_DB_5".Q AND NOT "P_TRIG".ARR[70];   // rising edge
   "P_TRIG".ARR[70] := "IEC_Timer_0_DB_5".Q;
   IF #_w1 THEN "HOOTER" := TRUE; END_IF;
END_REGION

REGION Network 72: EDI-501A PRODUCT OUT PRESSURE PT-504 HIGH
   RUNG wire#powerrail
      { S7_Templates := "SrcType := Int" } EQ_Contact(in1 := "INTERLOCK DB"."EDI PARAMETER BUFF"."PT-504 HIGH", in2 := 2)
      wire#w1
      Coil( "ALARM DB PLC 2"."EDI-501A PRODUCT OUT PRESSURE PT-504 HIGH" )
   END_RUNG
   RUNG wire#w1
      P_Trig( "P_TRIG".ARR[71] )
      S_Coil( "HOOTER" )
   END_RUNG
   // the same network as SCL:
   "ALARM DB PLC 2"."EDI-501A PRODUCT OUT PRESSURE PT-504 HIGH" := "INTERLOCK DB"."EDI PARAMETER BUFF"."PT-504 HIGH" = 2;
   #_w1 := "ALARM DB PLC 2"."EDI-501A PRODUCT OUT PRESSURE PT-504 HIGH" AND NOT "P_TRIG".ARR[71];   // rising edge
   "P_TRIG".ARR[71] := "ALARM DB PLC 2"."EDI-501A PRODUCT OUT PRESSURE PT-504 HIGH";
   IF #_w1 THEN "HOOTER" := TRUE; END_IF;
END_REGION

REGION Network 73: PT-504 HIGH_SET VALIDATION TIME OVER_(SYSTEM STOP)
   RUNG wire#powerrail
      Contact( "TIMING_SECS_DB_13".DONE )
      { S7_Templates := "time_type := Time" } "IEC_Timer_0_DB_6".TOF(pt := T#1S, et =>)
      wire#w1
      Coil( "ALARM DB PLC 2"."PT-504 HIGH_SET VALIDATION TIME OVER_(SYSTEM STOP)" )
   END_RUNG
   RUNG wire#w1
      P_Trig( "P_TRIG".ARR[72] )
      S_Coil( "HOOTER" )
   END_RUNG
   // the same network as SCL:
   "IEC_Timer_0_DB_6".TOF(IN := "TIMING_SECS_DB_13".DONE, PT := T#1S);
   "ALARM DB PLC 2"."PT-504 HIGH_SET VALIDATION TIME OVER_(SYSTEM STOP)" := "IEC_Timer_0_DB_6".Q;
   #_w1 := "IEC_Timer_0_DB_6".Q AND NOT "P_TRIG".ARR[72];   // rising edge
   "P_TRIG".ARR[72] := "IEC_Timer_0_DB_6".Q;
   IF #_w1 THEN "HOOTER" := TRUE; END_IF;
END_REGION

REGION Network 74: EDI-501A CONCENTRATE OUT PRESSURE PT-505 HIGH
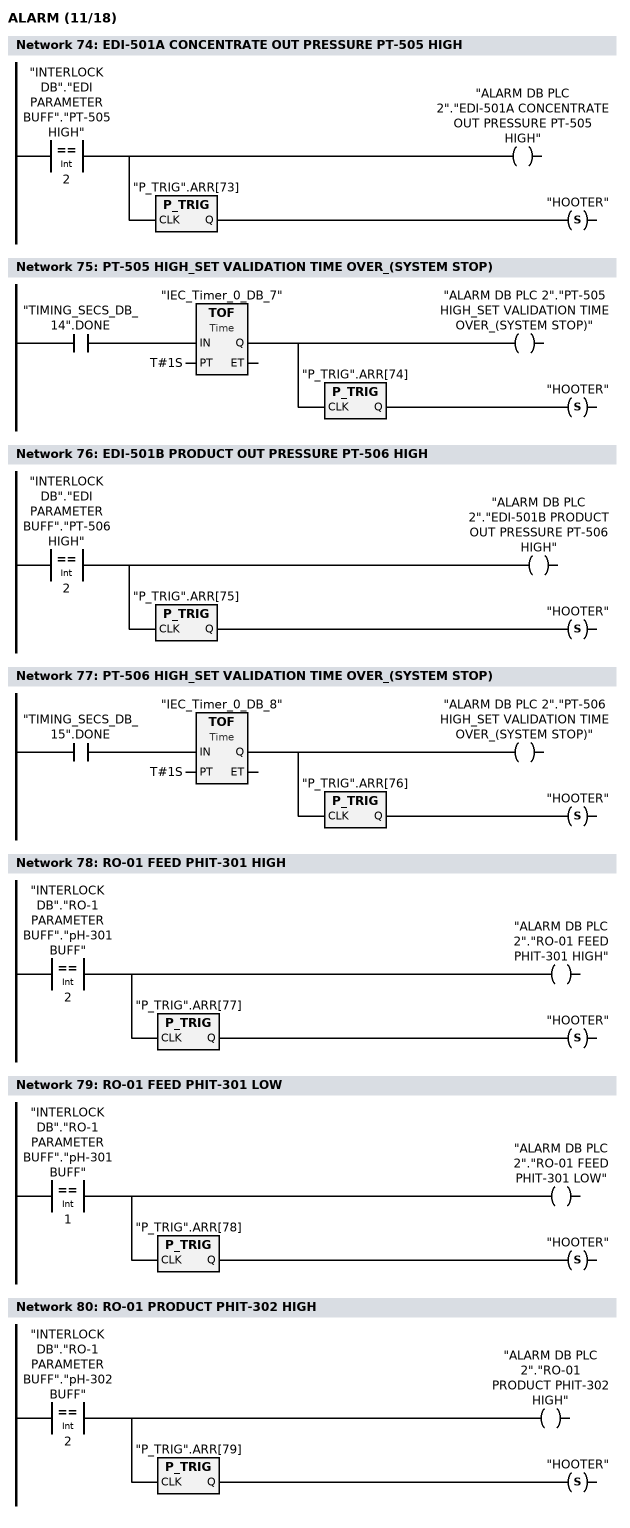
   RUNG wire#powerrail
      { S7_Templates := "SrcType := Int" } EQ_Contact(in1 := "INTERLOCK DB"."EDI PARAMETER BUFF"."PT-505 HIGH", in2 := 2)
      wire#w1
      Coil( "ALARM DB PLC 2"."EDI-501A CONCENTRATE OUT PRESSURE PT-505 HIGH" )
   END_RUNG
   RUNG wire#w1
      P_Trig( "P_TRIG".ARR[73] )
      S_Coil( "HOOTER" )
   END_RUNG
   // the same network as SCL:
   "ALARM DB PLC 2"."EDI-501A CONCENTRATE OUT PRESSURE PT-505 HIGH" := "INTERLOCK DB"."EDI PARAMETER BUFF"."PT-505 HIGH" = 2;
   #_w1 := "ALARM DB PLC 2"."EDI-501A CONCENTRATE OUT PRESSURE PT-505 HIGH" AND NOT "P_TRIG".ARR[73];   // rising edge
   "P_TRIG".ARR[73] := "ALARM DB PLC 2"."EDI-501A CONCENTRATE OUT PRESSURE PT-505 HIGH";
   IF #_w1 THEN "HOOTER" := TRUE; END_IF;
END_REGION

REGION Network 75: PT-505 HIGH_SET VALIDATION TIME OVER_(SYSTEM STOP)
   RUNG wire#powerrail
      Contact( "TIMING_SECS_DB_14".DONE )
      { S7_Templates := "time_type := Time" } "IEC_Timer_0_DB_7".TOF(pt := T#1S, et =>)
      wire#w1
      Coil( "ALARM DB PLC 2"."PT-505 HIGH_SET VALIDATION TIME OVER_(SYSTEM STOP)" )
   END_RUNG
   RUNG wire#w1
      P_Trig( "P_TRIG".ARR[74] )
      S_Coil( "HOOTER" )
   END_RUNG
   // the same network as SCL:
   "IEC_Timer_0_DB_7".TOF(IN := "TIMING_SECS_DB_14".DONE, PT := T#1S);
   "ALARM DB PLC 2"."PT-505 HIGH_SET VALIDATION TIME OVER_(SYSTEM STOP)" := "IEC_Timer_0_DB_7".Q;
   #_w1 := "IEC_Timer_0_DB_7".Q AND NOT "P_TRIG".ARR[74];   // rising edge
   "P_TRIG".ARR[74] := "IEC_Timer_0_DB_7".Q;
   IF #_w1 THEN "HOOTER" := TRUE; END_IF;
END_REGION

REGION Network 76: EDI-501B PRODUCT OUT PRESSURE PT-506 HIGH
   RUNG wire#powerrail
      { S7_Templates := "SrcType := Int" } EQ_Contact(in1 := "INTERLOCK DB"."EDI PARAMETER BUFF"."PT-506 HIGH", in2 := 2)
      wire#w1
      Coil( "ALARM DB PLC 2"."EDI-501B PRODUCT OUT PRESSURE PT-506 HIGH" )
   END_RUNG
   RUNG wire#w1
      P_Trig( "P_TRIG".ARR[75] )
      S_Coil( "HOOTER" )
   END_RUNG
   // the same network as SCL:
   "ALARM DB PLC 2"."EDI-501B PRODUCT OUT PRESSURE PT-506 HIGH" := "INTERLOCK DB"."EDI PARAMETER BUFF"."PT-506 HIGH" = 2;
   #_w1 := "ALARM DB PLC 2"."EDI-501B PRODUCT OUT PRESSURE PT-506 HIGH" AND NOT "P_TRIG".ARR[75];   // rising edge
   "P_TRIG".ARR[75] := "ALARM DB PLC 2"."EDI-501B PRODUCT OUT PRESSURE PT-506 HIGH";
   IF #_w1 THEN "HOOTER" := TRUE; END_IF;
END_REGION

REGION Network 77: PT-506 HIGH_SET VALIDATION TIME OVER_(SYSTEM STOP)
   RUNG wire#powerrail
      Contact( "TIMING_SECS_DB_15".DONE )
      { S7_Templates := "time_type := Time" } "IEC_Timer_0_DB_8".TOF(pt := T#1S, et =>)
      wire#w1
      Coil( "ALARM DB PLC 2"."PT-506 HIGH_SET VALIDATION TIME OVER_(SYSTEM STOP)" )
   END_RUNG
   RUNG wire#w1
      P_Trig( "P_TRIG".ARR[76] )
      S_Coil( "HOOTER" )
   END_RUNG
   // the same network as SCL:
   "IEC_Timer_0_DB_8".TOF(IN := "TIMING_SECS_DB_15".DONE, PT := T#1S);
   "ALARM DB PLC 2"."PT-506 HIGH_SET VALIDATION TIME OVER_(SYSTEM STOP)" := "IEC_Timer_0_DB_8".Q;
   #_w1 := "IEC_Timer_0_DB_8".Q AND NOT "P_TRIG".ARR[76];   // rising edge
   "P_TRIG".ARR[76] := "IEC_Timer_0_DB_8".Q;
   IF #_w1 THEN "HOOTER" := TRUE; END_IF;
END_REGION

REGION Network 78: RO-01 FEED PHIT-301 HIGH
   RUNG wire#powerrail
      { S7_Templates := "SrcType := Int" } EQ_Contact(in1 := "INTERLOCK DB"."RO-1 PARAMETER BUFF"."pH-301 BUFF", in2 := 2)
      wire#w1
      Coil( "ALARM DB PLC 2"."RO-01 FEED PHIT-301 HIGH" )
   END_RUNG
   RUNG wire#w1
      P_Trig( "P_TRIG".ARR[77] )
      S_Coil( "HOOTER" )
   END_RUNG
   // the same network as SCL:
   "ALARM DB PLC 2"."RO-01 FEED PHIT-301 HIGH" := "INTERLOCK DB"."RO-1 PARAMETER BUFF"."pH-301 BUFF" = 2;
   #_w1 := "ALARM DB PLC 2"."RO-01 FEED PHIT-301 HIGH" AND NOT "P_TRIG".ARR[77];   // rising edge
   "P_TRIG".ARR[77] := "ALARM DB PLC 2"."RO-01 FEED PHIT-301 HIGH";
   IF #_w1 THEN "HOOTER" := TRUE; END_IF;
END_REGION

REGION Network 79: RO-01 FEED PHIT-301 LOW
   RUNG wire#powerrail
      { S7_Templates := "SrcType := Int" } EQ_Contact(in1 := "INTERLOCK DB"."RO-1 PARAMETER BUFF"."pH-301 BUFF", in2 := 1)
      wire#w1
      Coil( "ALARM DB PLC 2"."RO-01 FEED PHIT-301 LOW" )
   END_RUNG
   RUNG wire#w1
      P_Trig( "P_TRIG".ARR[78] )
      S_Coil( "HOOTER" )
   END_RUNG
   // the same network as SCL:
   "ALARM DB PLC 2"."RO-01 FEED PHIT-301 LOW" := "INTERLOCK DB"."RO-1 PARAMETER BUFF"."pH-301 BUFF" = 1;
   #_w1 := "ALARM DB PLC 2"."RO-01 FEED PHIT-301 LOW" AND NOT "P_TRIG".ARR[78];   // rising edge
   "P_TRIG".ARR[78] := "ALARM DB PLC 2"."RO-01 FEED PHIT-301 LOW";
   IF #_w1 THEN "HOOTER" := TRUE; END_IF;
END_REGION

REGION Network 80: RO-01 PRODUCT PHIT-302 HIGH
   RUNG wire#powerrail
      { S7_Templates := "SrcType := Int" } EQ_Contact(in1 := "INTERLOCK DB"."RO-1 PARAMETER BUFF"."pH-302 BUFF", in2 := 2)
      wire#w1
      Coil( "ALARM DB PLC 2"."RO-01 PRODUCT PHIT-302 HIGH" )
   END_RUNG
   RUNG wire#w1
      P_Trig( "P_TRIG".ARR[79] )
      S_Coil( "HOOTER" )
   END_RUNG
   // the same network as SCL:
   "ALARM DB PLC 2"."RO-01 PRODUCT PHIT-302 HIGH" := "INTERLOCK DB"."RO-1 PARAMETER BUFF"."pH-302 BUFF" = 2;
   #_w1 := "ALARM DB PLC 2"."RO-01 PRODUCT PHIT-302 HIGH" AND NOT "P_TRIG".ARR[79];   // rising edge
   "P_TRIG".ARR[79] := "ALARM DB PLC 2"."RO-01 PRODUCT PHIT-302 HIGH";
   IF #_w1 THEN "HOOTER" := TRUE; END_IF;
END_REGION

REGION Network 81: RO-01 PRODUCT PHIT-302 LOW
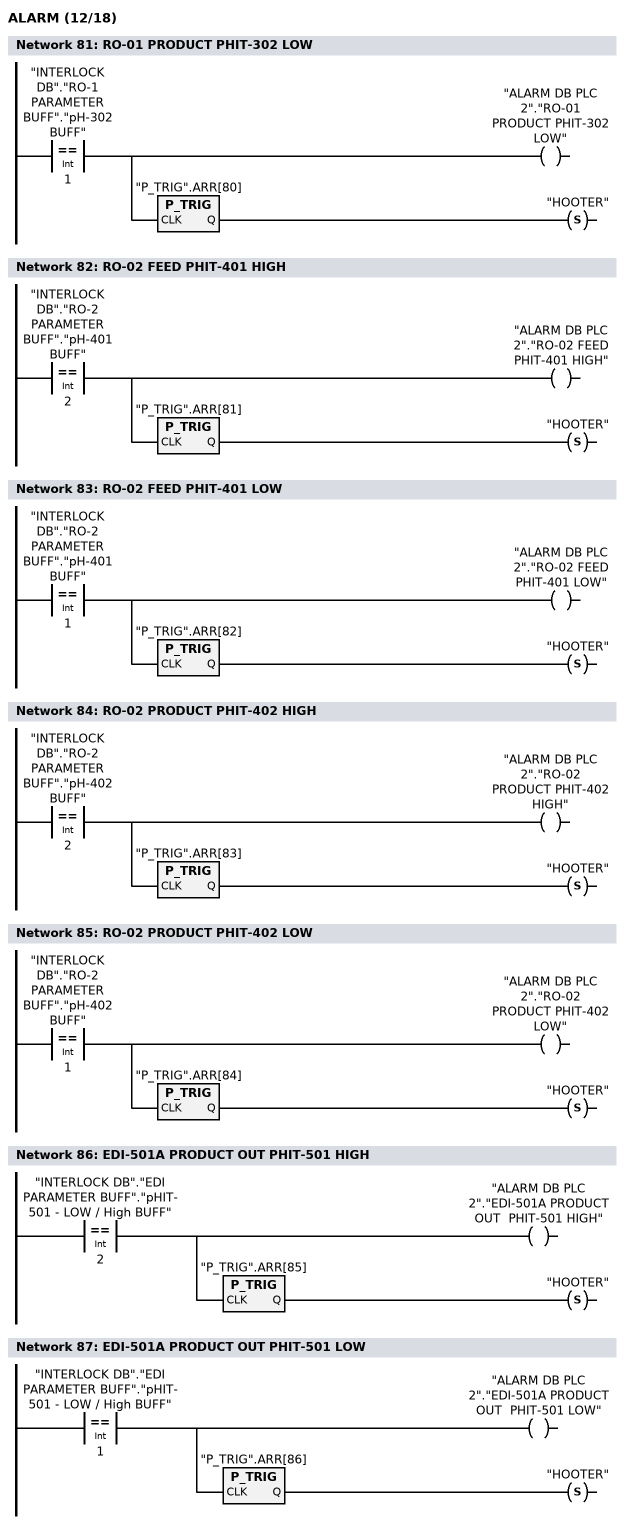
   RUNG wire#powerrail
      { S7_Templates := "SrcType := Int" } EQ_Contact(in1 := "INTERLOCK DB"."RO-1 PARAMETER BUFF"."pH-302 BUFF", in2 := 1)
      wire#w1
      Coil( "ALARM DB PLC 2"."RO-01 PRODUCT PHIT-302 LOW" )
   END_RUNG
   RUNG wire#w1
      P_Trig( "P_TRIG".ARR[80] )
      S_Coil( "HOOTER" )
   END_RUNG
   // the same network as SCL:
   "ALARM DB PLC 2"."RO-01 PRODUCT PHIT-302 LOW" := "INTERLOCK DB"."RO-1 PARAMETER BUFF"."pH-302 BUFF" = 1;
   #_w1 := "ALARM DB PLC 2"."RO-01 PRODUCT PHIT-302 LOW" AND NOT "P_TRIG".ARR[80];   // rising edge
   "P_TRIG".ARR[80] := "ALARM DB PLC 2"."RO-01 PRODUCT PHIT-302 LOW";
   IF #_w1 THEN "HOOTER" := TRUE; END_IF;
END_REGION

REGION Network 82: RO-02 FEED PHIT-401 HIGH
   RUNG wire#powerrail
      { S7_Templates := "SrcType := Int" } EQ_Contact(in1 := "INTERLOCK DB"."RO-2 PARAMETER BUFF"."pH-401 BUFF", in2 := 2)
      wire#w1
      Coil( "ALARM DB PLC 2"."RO-02 FEED PHIT-401 HIGH" )
   END_RUNG
   RUNG wire#w1
      P_Trig( "P_TRIG".ARR[81] )
      S_Coil( "HOOTER" )
   END_RUNG
   // the same network as SCL:
   "ALARM DB PLC 2"."RO-02 FEED PHIT-401 HIGH" := "INTERLOCK DB"."RO-2 PARAMETER BUFF"."pH-401 BUFF" = 2;
   #_w1 := "ALARM DB PLC 2"."RO-02 FEED PHIT-401 HIGH" AND NOT "P_TRIG".ARR[81];   // rising edge
   "P_TRIG".ARR[81] := "ALARM DB PLC 2"."RO-02 FEED PHIT-401 HIGH";
   IF #_w1 THEN "HOOTER" := TRUE; END_IF;
END_REGION

REGION Network 83: RO-02 FEED PHIT-401 LOW
   RUNG wire#powerrail
      { S7_Templates := "SrcType := Int" } EQ_Contact(in1 := "INTERLOCK DB"."RO-2 PARAMETER BUFF"."pH-401 BUFF", in2 := 1)
      wire#w1
      Coil( "ALARM DB PLC 2"."RO-02 FEED PHIT-401 LOW" )
   END_RUNG
   RUNG wire#w1
      P_Trig( "P_TRIG".ARR[82] )
      S_Coil( "HOOTER" )
   END_RUNG
   // the same network as SCL:
   "ALARM DB PLC 2"."RO-02 FEED PHIT-401 LOW" := "INTERLOCK DB"."RO-2 PARAMETER BUFF"."pH-401 BUFF" = 1;
   #_w1 := "ALARM DB PLC 2"."RO-02 FEED PHIT-401 LOW" AND NOT "P_TRIG".ARR[82];   // rising edge
   "P_TRIG".ARR[82] := "ALARM DB PLC 2"."RO-02 FEED PHIT-401 LOW";
   IF #_w1 THEN "HOOTER" := TRUE; END_IF;
END_REGION

REGION Network 84: RO-02 PRODUCT PHIT-402 HIGH
   RUNG wire#powerrail
      { S7_Templates := "SrcType := Int" } EQ_Contact(in1 := "INTERLOCK DB"."RO-2 PARAMETER BUFF"."pH-402 BUFF", in2 := 2)
      wire#w1
      Coil( "ALARM DB PLC 2"."RO-02 PRODUCT PHIT-402 HIGH" )
   END_RUNG
   RUNG wire#w1
      P_Trig( "P_TRIG".ARR[83] )
      S_Coil( "HOOTER" )
   END_RUNG
   // the same network as SCL:
   "ALARM DB PLC 2"."RO-02 PRODUCT PHIT-402 HIGH" := "INTERLOCK DB"."RO-2 PARAMETER BUFF"."pH-402 BUFF" = 2;
   #_w1 := "ALARM DB PLC 2"."RO-02 PRODUCT PHIT-402 HIGH" AND NOT "P_TRIG".ARR[83];   // rising edge
   "P_TRIG".ARR[83] := "ALARM DB PLC 2"."RO-02 PRODUCT PHIT-402 HIGH";
   IF #_w1 THEN "HOOTER" := TRUE; END_IF;
END_REGION

REGION Network 85: RO-02 PRODUCT PHIT-402 LOW
   RUNG wire#powerrail
      { S7_Templates := "SrcType := Int" } EQ_Contact(in1 := "INTERLOCK DB"."RO-2 PARAMETER BUFF"."pH-402 BUFF", in2 := 1)
      wire#w1
      Coil( "ALARM DB PLC 2"."RO-02 PRODUCT PHIT-402 LOW" )
   END_RUNG
   RUNG wire#w1
      P_Trig( "P_TRIG".ARR[84] )
      S_Coil( "HOOTER" )
   END_RUNG
   // the same network as SCL:
   "ALARM DB PLC 2"."RO-02 PRODUCT PHIT-402 LOW" := "INTERLOCK DB"."RO-2 PARAMETER BUFF"."pH-402 BUFF" = 1;
   #_w1 := "ALARM DB PLC 2"."RO-02 PRODUCT PHIT-402 LOW" AND NOT "P_TRIG".ARR[84];   // rising edge
   "P_TRIG".ARR[84] := "ALARM DB PLC 2"."RO-02 PRODUCT PHIT-402 LOW";
   IF #_w1 THEN "HOOTER" := TRUE; END_IF;
END_REGION

REGION Network 86: EDI-501A PRODUCT OUT PHIT-501 HIGH
   RUNG wire#powerrail
      { S7_Templates := "SrcType := Int" } EQ_Contact(in1 := "INTERLOCK DB"."EDI PARAMETER BUFF"."pHIT-501 - LOW / High BUFF", in2 := 2)
      wire#w1
      Coil( "ALARM DB PLC 2"."EDI-501A PRODUCT OUT  PHIT-501 HIGH" )
   END_RUNG
   RUNG wire#w1
      P_Trig( "P_TRIG".ARR[85] )
      S_Coil( "HOOTER" )
   END_RUNG
   // the same network as SCL:
   "ALARM DB PLC 2"."EDI-501A PRODUCT OUT  PHIT-501 HIGH" := "INTERLOCK DB"."EDI PARAMETER BUFF"."pHIT-501 - LOW / High BUFF" = 2;
   #_w1 := "ALARM DB PLC 2"."EDI-501A PRODUCT OUT  PHIT-501 HIGH" AND NOT "P_TRIG".ARR[85];   // rising edge
   "P_TRIG".ARR[85] := "ALARM DB PLC 2"."EDI-501A PRODUCT OUT  PHIT-501 HIGH";
   IF #_w1 THEN "HOOTER" := TRUE; END_IF;
END_REGION

REGION Network 87: EDI-501A PRODUCT OUT PHIT-501 LOW
   RUNG wire#powerrail
      { S7_Templates := "SrcType := Int" } EQ_Contact(in1 := "INTERLOCK DB"."EDI PARAMETER BUFF"."pHIT-501 - LOW / High BUFF", in2 := 1)
      wire#w1
      Coil( "ALARM DB PLC 2"."EDI-501A PRODUCT OUT  PHIT-501 LOW" )
   END_RUNG
   RUNG wire#w1
      P_Trig( "P_TRIG".ARR[86] )
      S_Coil( "HOOTER" )
   END_RUNG
   // the same network as SCL:
   "ALARM DB PLC 2"."EDI-501A PRODUCT OUT  PHIT-501 LOW" := "INTERLOCK DB"."EDI PARAMETER BUFF"."pHIT-501 - LOW / High BUFF" = 1;
   #_w1 := "ALARM DB PLC 2"."EDI-501A PRODUCT OUT  PHIT-501 LOW" AND NOT "P_TRIG".ARR[86];   // rising edge
   "P_TRIG".ARR[86] := "ALARM DB PLC 2"."EDI-501A PRODUCT OUT  PHIT-501 LOW";
   IF #_w1 THEN "HOOTER" := TRUE; END_IF;
END_REGION

REGION Network 88: EDI-501B PRODUCT OUT PHIT-502 HIGH
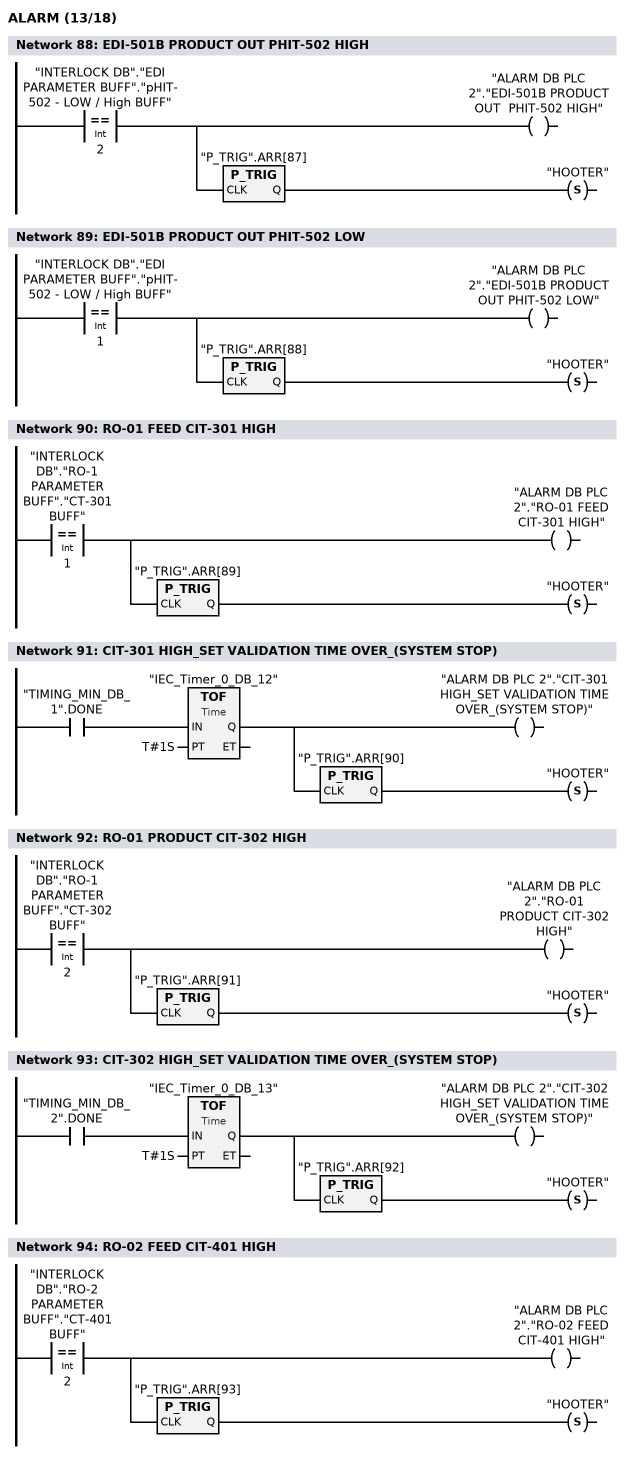
   RUNG wire#powerrail
      { S7_Templates := "SrcType := Int" } EQ_Contact(in1 := "INTERLOCK DB"."EDI PARAMETER BUFF"."pHIT-502 - LOW / High BUFF", in2 := 2)
      wire#w1
      Coil( "ALARM DB PLC 2"."EDI-501B PRODUCT OUT  PHIT-502 HIGH" )
   END_RUNG
   RUNG wire#w1
      P_Trig( "P_TRIG".ARR[87] )
      S_Coil( "HOOTER" )
   END_RUNG
   // the same network as SCL:
   "ALARM DB PLC 2"."EDI-501B PRODUCT OUT  PHIT-502 HIGH" := "INTERLOCK DB"."EDI PARAMETER BUFF"."pHIT-502 - LOW / High BUFF" = 2;
   #_w1 := "ALARM DB PLC 2"."EDI-501B PRODUCT OUT  PHIT-502 HIGH" AND NOT "P_TRIG".ARR[87];   // rising edge
   "P_TRIG".ARR[87] := "ALARM DB PLC 2"."EDI-501B PRODUCT OUT  PHIT-502 HIGH";
   IF #_w1 THEN "HOOTER" := TRUE; END_IF;
END_REGION

REGION Network 89: EDI-501B PRODUCT OUT PHIT-502 LOW
   RUNG wire#powerrail
      { S7_Templates := "SrcType := Int" } EQ_Contact(in1 := "INTERLOCK DB"."EDI PARAMETER BUFF"."pHIT-502 - LOW / High BUFF", in2 := 1)
      wire#w1
      Coil( "ALARM DB PLC 2"."EDI-501B PRODUCT OUT PHIT-502 LOW" )
   END_RUNG
   RUNG wire#w1
      P_Trig( "P_TRIG".ARR[88] )
      S_Coil( "HOOTER" )
   END_RUNG
   // the same network as SCL:
   "ALARM DB PLC 2"."EDI-501B PRODUCT OUT PHIT-502 LOW" := "INTERLOCK DB"."EDI PARAMETER BUFF"."pHIT-502 - LOW / High BUFF" = 1;
   #_w1 := "ALARM DB PLC 2"."EDI-501B PRODUCT OUT PHIT-502 LOW" AND NOT "P_TRIG".ARR[88];   // rising edge
   "P_TRIG".ARR[88] := "ALARM DB PLC 2"."EDI-501B PRODUCT OUT PHIT-502 LOW";
   IF #_w1 THEN "HOOTER" := TRUE; END_IF;
END_REGION

REGION Network 90: RO-01 FEED CIT-301 HIGH
   RUNG wire#powerrail
      { S7_Templates := "SrcType := Int" } EQ_Contact(in1 := "INTERLOCK DB"."RO-1 PARAMETER BUFF"."CT-301 BUFF", in2 := 1)
      wire#w1
      Coil( "ALARM DB PLC 2"."RO-01 FEED CIT-301 HIGH" )
   END_RUNG
   RUNG wire#w1
      P_Trig( "P_TRIG".ARR[89] )
      S_Coil( "HOOTER" )
   END_RUNG
   // the same network as SCL:
   "ALARM DB PLC 2"."RO-01 FEED CIT-301 HIGH" := "INTERLOCK DB"."RO-1 PARAMETER BUFF"."CT-301 BUFF" = 1;
   #_w1 := "ALARM DB PLC 2"."RO-01 FEED CIT-301 HIGH" AND NOT "P_TRIG".ARR[89];   // rising edge
   "P_TRIG".ARR[89] := "ALARM DB PLC 2"."RO-01 FEED CIT-301 HIGH";
   IF #_w1 THEN "HOOTER" := TRUE; END_IF;
END_REGION

REGION Network 91: CIT-301 HIGH_SET VALIDATION TIME OVER_(SYSTEM STOP)
   RUNG wire#powerrail
      Contact( "TIMING_MIN_DB_1".DONE )
      { S7_Templates := "time_type := Time" } "IEC_Timer_0_DB_12".TOF(pt := T#1S, et =>)
      wire#w1
      Coil( "ALARM DB PLC 2"."CIT-301 HIGH_SET VALIDATION TIME OVER_(SYSTEM STOP)" )
   END_RUNG
   RUNG wire#w1
      P_Trig( "P_TRIG".ARR[90] )
      S_Coil( "HOOTER" )
   END_RUNG
   // the same network as SCL:
   "IEC_Timer_0_DB_12".TOF(IN := "TIMING_MIN_DB_1".DONE, PT := T#1S);
   "ALARM DB PLC 2"."CIT-301 HIGH_SET VALIDATION TIME OVER_(SYSTEM STOP)" := "IEC_Timer_0_DB_12".Q;
   #_w1 := "IEC_Timer_0_DB_12".Q AND NOT "P_TRIG".ARR[90];   // rising edge
   "P_TRIG".ARR[90] := "IEC_Timer_0_DB_12".Q;
   IF #_w1 THEN "HOOTER" := TRUE; END_IF;
END_REGION

REGION Network 92: RO-01 PRODUCT CIT-302 HIGH
   RUNG wire#powerrail
      { S7_Templates := "SrcType := Int" } EQ_Contact(in1 := "INTERLOCK DB"."RO-1 PARAMETER BUFF"."CT-302 BUFF", in2 := 2)
      wire#w1
      Coil( "ALARM DB PLC 2"."RO-01 PRODUCT CIT-302 HIGH" )
   END_RUNG
   RUNG wire#w1
      P_Trig( "P_TRIG".ARR[91] )
      S_Coil( "HOOTER" )
   END_RUNG
   // the same network as SCL:
   "ALARM DB PLC 2"."RO-01 PRODUCT CIT-302 HIGH" := "INTERLOCK DB"."RO-1 PARAMETER BUFF"."CT-302 BUFF" = 2;
   #_w1 := "ALARM DB PLC 2"."RO-01 PRODUCT CIT-302 HIGH" AND NOT "P_TRIG".ARR[91];   // rising edge
   "P_TRIG".ARR[91] := "ALARM DB PLC 2"."RO-01 PRODUCT CIT-302 HIGH";
   IF #_w1 THEN "HOOTER" := TRUE; END_IF;
END_REGION

REGION Network 93: CIT-302 HIGH_SET VALIDATION TIME OVER_(SYSTEM STOP)
   RUNG wire#powerrail
      Contact( "TIMING_MIN_DB_2".DONE )
      { S7_Templates := "time_type := Time" } "IEC_Timer_0_DB_13".TOF(pt := T#1S, et =>)
      wire#w1
      Coil( "ALARM DB PLC 2"."CIT-302 HIGH_SET VALIDATION TIME OVER_(SYSTEM STOP)" )
   END_RUNG
   RUNG wire#w1
      P_Trig( "P_TRIG".ARR[92] )
      S_Coil( "HOOTER" )
   END_RUNG
   // the same network as SCL:
   "IEC_Timer_0_DB_13".TOF(IN := "TIMING_MIN_DB_2".DONE, PT := T#1S);
   "ALARM DB PLC 2"."CIT-302 HIGH_SET VALIDATION TIME OVER_(SYSTEM STOP)" := "IEC_Timer_0_DB_13".Q;
   #_w1 := "IEC_Timer_0_DB_13".Q AND NOT "P_TRIG".ARR[92];   // rising edge
   "P_TRIG".ARR[92] := "IEC_Timer_0_DB_13".Q;
   IF #_w1 THEN "HOOTER" := TRUE; END_IF;
END_REGION

REGION Network 94: RO-02 FEED CIT-401 HIGH
   RUNG wire#powerrail
      { S7_Templates := "SrcType := Int" } EQ_Contact(in1 := "INTERLOCK DB"."RO-2 PARAMETER BUFF"."CT-401 BUFF", in2 := 2)
      wire#w1
      Coil( "ALARM DB PLC 2"."RO-02 FEED CIT-401 HIGH" )
   END_RUNG
   RUNG wire#w1
      P_Trig( "P_TRIG".ARR[93] )
      S_Coil( "HOOTER" )
   END_RUNG
   // the same network as SCL:
   "ALARM DB PLC 2"."RO-02 FEED CIT-401 HIGH" := "INTERLOCK DB"."RO-2 PARAMETER BUFF"."CT-401 BUFF" = 2;
   #_w1 := "ALARM DB PLC 2"."RO-02 FEED CIT-401 HIGH" AND NOT "P_TRIG".ARR[93];   // rising edge
   "P_TRIG".ARR[93] := "ALARM DB PLC 2"."RO-02 FEED CIT-401 HIGH";
   IF #_w1 THEN "HOOTER" := TRUE; END_IF;
END_REGION

REGION Network 95: CIT-401 HIGH_SET VALIDATION TIME OVER_(SYSTEM STOP)
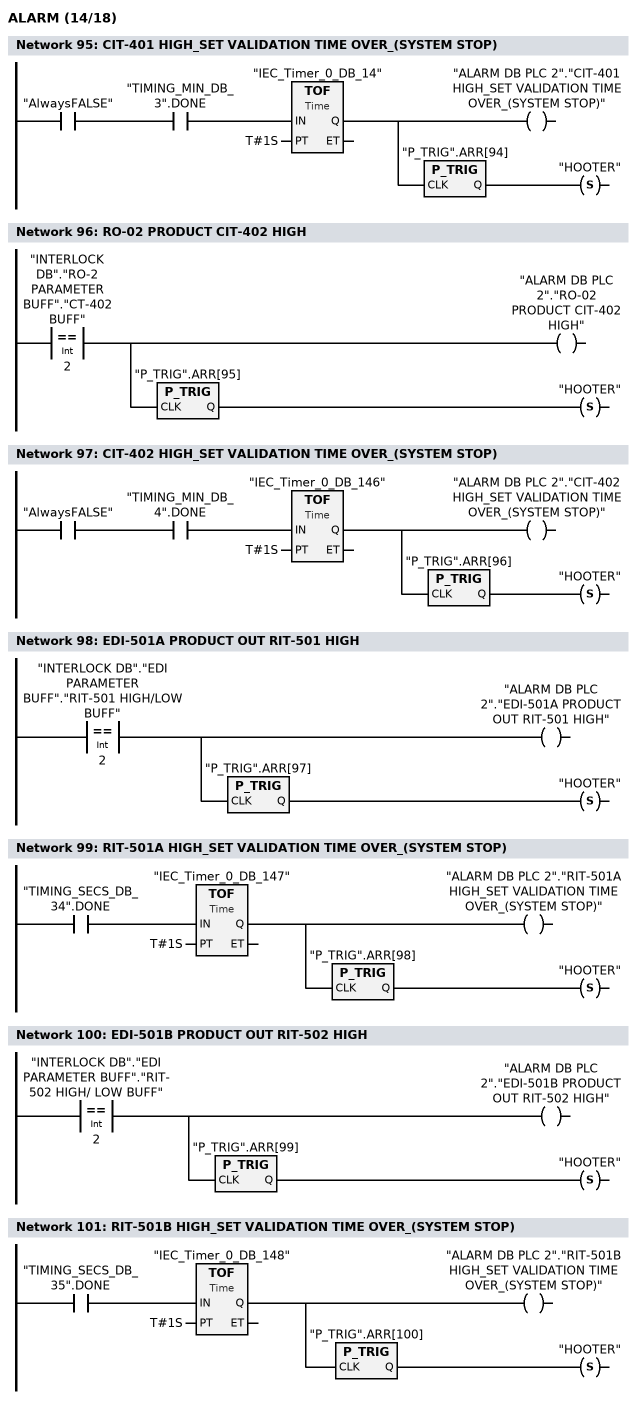
   RUNG wire#powerrail
      Contact( "AlwaysFALSE" )
      Contact( "TIMING_MIN_DB_3".DONE )
      { S7_Templates := "time_type := Time" } "IEC_Timer_0_DB_14".TOF(pt := T#1S, et =>)
      wire#w1
      Coil( "ALARM DB PLC 2"."CIT-401 HIGH_SET VALIDATION TIME OVER_(SYSTEM STOP)" )
   END_RUNG
   RUNG wire#w1
      P_Trig( "P_TRIG".ARR[94] )
      S_Coil( "HOOTER" )
   END_RUNG
   // the same network as SCL:
   "IEC_Timer_0_DB_14".TOF(IN := "AlwaysFALSE" AND "TIMING_MIN_DB_3".DONE, PT := T#1S);
   "ALARM DB PLC 2"."CIT-401 HIGH_SET VALIDATION TIME OVER_(SYSTEM STOP)" := "IEC_Timer_0_DB_14".Q;
   #_w1 := "IEC_Timer_0_DB_14".Q AND NOT "P_TRIG".ARR[94];   // rising edge
   "P_TRIG".ARR[94] := "IEC_Timer_0_DB_14".Q;
   IF #_w1 THEN "HOOTER" := TRUE; END_IF;
END_REGION

REGION Network 96: RO-02 PRODUCT CIT-402 HIGH
   RUNG wire#powerrail
      { S7_Templates := "SrcType := Int" } EQ_Contact(in1 := "INTERLOCK DB"."RO-2 PARAMETER BUFF"."CT-402 BUFF", in2 := 2)
      wire#w1
      Coil( "ALARM DB PLC 2"."RO-02 PRODUCT CIT-402 HIGH" )
   END_RUNG
   RUNG wire#w1
      P_Trig( "P_TRIG".ARR[95] )
      S_Coil( "HOOTER" )
   END_RUNG
   // the same network as SCL:
   "ALARM DB PLC 2"."RO-02 PRODUCT CIT-402 HIGH" := "INTERLOCK DB"."RO-2 PARAMETER BUFF"."CT-402 BUFF" = 2;
   #_w1 := "ALARM DB PLC 2"."RO-02 PRODUCT CIT-402 HIGH" AND NOT "P_TRIG".ARR[95];   // rising edge
   "P_TRIG".ARR[95] := "ALARM DB PLC 2"."RO-02 PRODUCT CIT-402 HIGH";
   IF #_w1 THEN "HOOTER" := TRUE; END_IF;
END_REGION

REGION Network 97: CIT-402 HIGH_SET VALIDATION TIME OVER_(SYSTEM STOP)
   RUNG wire#powerrail
      Contact( "AlwaysFALSE" )
      Contact( "TIMING_MIN_DB_4".DONE )
      { S7_Templates := "time_type := Time" } "IEC_Timer_0_DB_146".TOF(pt := T#1S, et =>)
      wire#w1
      Coil( "ALARM DB PLC 2"."CIT-402 HIGH_SET VALIDATION TIME OVER_(SYSTEM STOP)" )
   END_RUNG
   RUNG wire#w1
      P_Trig( "P_TRIG".ARR[96] )
      S_Coil( "HOOTER" )
   END_RUNG
   // the same network as SCL:
   "IEC_Timer_0_DB_146".TOF(IN := "AlwaysFALSE" AND "TIMING_MIN_DB_4".DONE, PT := T#1S);
   "ALARM DB PLC 2"."CIT-402 HIGH_SET VALIDATION TIME OVER_(SYSTEM STOP)" := "IEC_Timer_0_DB_146".Q;
   #_w1 := "IEC_Timer_0_DB_146".Q AND NOT "P_TRIG".ARR[96];   // rising edge
   "P_TRIG".ARR[96] := "IEC_Timer_0_DB_146".Q;
   IF #_w1 THEN "HOOTER" := TRUE; END_IF;
END_REGION

REGION Network 98: EDI-501A PRODUCT OUT RIT-501 HIGH
   RUNG wire#powerrail
      { S7_Templates := "SrcType := Int" } EQ_Contact(in1 := "INTERLOCK DB"."EDI PARAMETER BUFF"."RIT-501 HIGH/LOW BUFF", in2 := 2)
      wire#w1
      Coil( "ALARM DB PLC 2"."EDI-501A PRODUCT OUT RIT-501 HIGH" )
   END_RUNG
   RUNG wire#w1
      P_Trig( "P_TRIG".ARR[97] )
      S_Coil( "HOOTER" )
   END_RUNG
   // the same network as SCL:
   "ALARM DB PLC 2"."EDI-501A PRODUCT OUT RIT-501 HIGH" := "INTERLOCK DB"."EDI PARAMETER BUFF"."RIT-501 HIGH/LOW BUFF" = 2;
   #_w1 := "ALARM DB PLC 2"."EDI-501A PRODUCT OUT RIT-501 HIGH" AND NOT "P_TRIG".ARR[97];   // rising edge
   "P_TRIG".ARR[97] := "ALARM DB PLC 2"."EDI-501A PRODUCT OUT RIT-501 HIGH";
   IF #_w1 THEN "HOOTER" := TRUE; END_IF;
END_REGION

REGION Network 99: RIT-501A HIGH_SET VALIDATION TIME OVER_(SYSTEM STOP)
   RUNG wire#powerrail
      Contact( "TIMING_SECS_DB_34".DONE )
      { S7_Templates := "time_type := Time" } "IEC_Timer_0_DB_147".TOF(pt := T#1S, et =>)
      wire#w1
      Coil( "ALARM DB PLC 2"."RIT-501A HIGH_SET VALIDATION TIME OVER_(SYSTEM STOP)" )
   END_RUNG
   RUNG wire#w1
      P_Trig( "P_TRIG".ARR[98] )
      S_Coil( "HOOTER" )
   END_RUNG
   // the same network as SCL:
   "IEC_Timer_0_DB_147".TOF(IN := "TIMING_SECS_DB_34".DONE, PT := T#1S);
   "ALARM DB PLC 2"."RIT-501A HIGH_SET VALIDATION TIME OVER_(SYSTEM STOP)" := "IEC_Timer_0_DB_147".Q;
   #_w1 := "IEC_Timer_0_DB_147".Q AND NOT "P_TRIG".ARR[98];   // rising edge
   "P_TRIG".ARR[98] := "IEC_Timer_0_DB_147".Q;
   IF #_w1 THEN "HOOTER" := TRUE; END_IF;
END_REGION

REGION Network 100: EDI-501B PRODUCT OUT RIT-502 HIGH
   RUNG wire#powerrail
      { S7_Templates := "SrcType := Int" } EQ_Contact(in1 := "INTERLOCK DB"."EDI PARAMETER BUFF"."RIT-502 HIGH/ LOW BUFF", in2 := 2)
      wire#w1
      Coil( "ALARM DB PLC 2"."EDI-501B PRODUCT OUT RIT-502 HIGH" )
   END_RUNG
   RUNG wire#w1
      P_Trig( "P_TRIG".ARR[99] )
      S_Coil( "HOOTER" )
   END_RUNG
   // the same network as SCL:
   "ALARM DB PLC 2"."EDI-501B PRODUCT OUT RIT-502 HIGH" := "INTERLOCK DB"."EDI PARAMETER BUFF"."RIT-502 HIGH/ LOW BUFF" = 2;
   #_w1 := "ALARM DB PLC 2"."EDI-501B PRODUCT OUT RIT-502 HIGH" AND NOT "P_TRIG".ARR[99];   // rising edge
   "P_TRIG".ARR[99] := "ALARM DB PLC 2"."EDI-501B PRODUCT OUT RIT-502 HIGH";
   IF #_w1 THEN "HOOTER" := TRUE; END_IF;
END_REGION

REGION Network 101: RIT-501B HIGH_SET VALIDATION TIME OVER_(SYSTEM STOP)
   RUNG wire#powerrail
      Contact( "TIMING_SECS_DB_35".DONE )
      { S7_Templates := "time_type := Time" } "IEC_Timer_0_DB_148".TOF(pt := T#1S, et =>)
      wire#w1
      Coil( "ALARM DB PLC 2"."RIT-501B HIGH_SET VALIDATION TIME OVER_(SYSTEM STOP)" )
   END_RUNG
   RUNG wire#w1
      P_Trig( "P_TRIG".ARR[100] )
      S_Coil( "HOOTER" )
   END_RUNG
   // the same network as SCL:
   "IEC_Timer_0_DB_148".TOF(IN := "TIMING_SECS_DB_35".DONE, PT := T#1S);
   "ALARM DB PLC 2"."RIT-501B HIGH_SET VALIDATION TIME OVER_(SYSTEM STOP)" := "IEC_Timer_0_DB_148".Q;
   #_w1 := "IEC_Timer_0_DB_148".Q AND NOT "P_TRIG".ARR[100];   // rising edge
   "P_TRIG".ARR[100] := "IEC_Timer_0_DB_148".Q;
   IF #_w1 THEN "HOOTER" := TRUE; END_IF;
END_REGION

REGION Network 102: ORP-301 HIGH
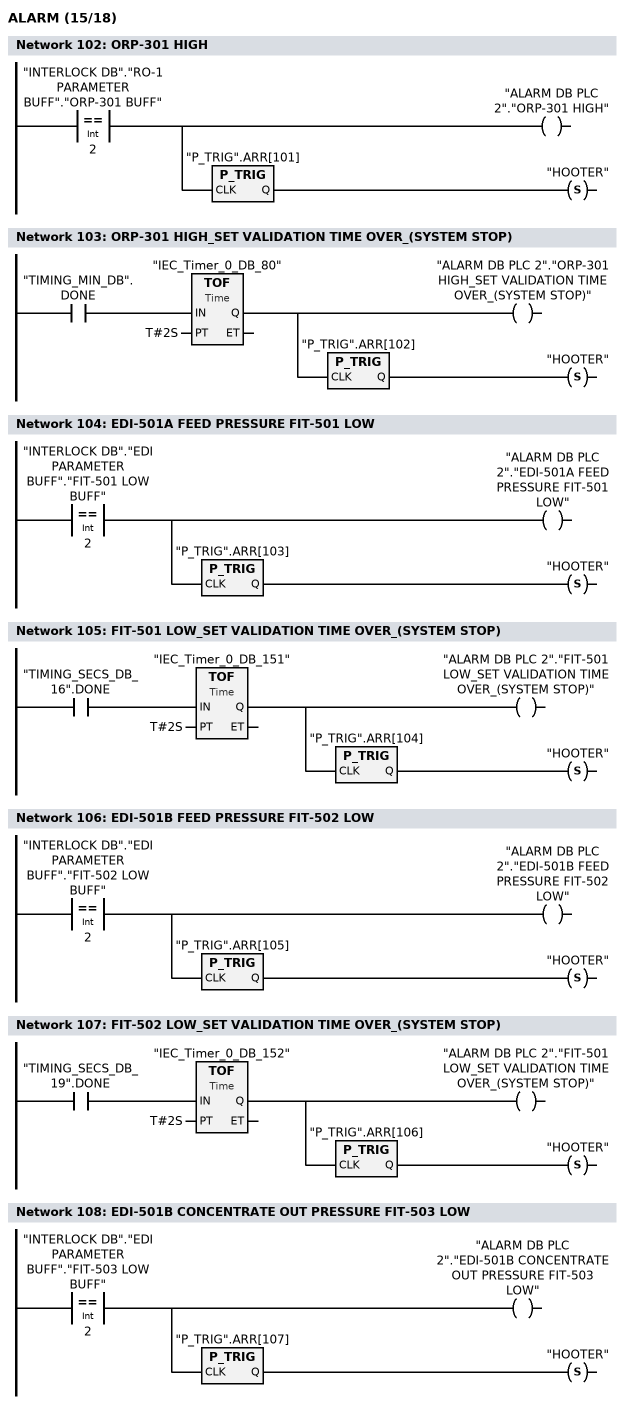
   RUNG wire#powerrail
      { S7_Templates := "SrcType := Int" } EQ_Contact(in1 := "INTERLOCK DB"."RO-1 PARAMETER BUFF"."ORP-301 BUFF", in2 := 2)
      wire#w1
      Coil( "ALARM DB PLC 2"."ORP-301 HIGH" )
   END_RUNG
   RUNG wire#w1
      P_Trig( "P_TRIG".ARR[101] )
      S_Coil( "HOOTER" )
   END_RUNG
   // the same network as SCL:
   "ALARM DB PLC 2"."ORP-301 HIGH" := "INTERLOCK DB"."RO-1 PARAMETER BUFF"."ORP-301 BUFF" = 2;
   #_w1 := "ALARM DB PLC 2"."ORP-301 HIGH" AND NOT "P_TRIG".ARR[101];   // rising edge
   "P_TRIG".ARR[101] := "ALARM DB PLC 2"."ORP-301 HIGH";
   IF #_w1 THEN "HOOTER" := TRUE; END_IF;
END_REGION

REGION Network 103: ORP-301 HIGH_SET VALIDATION TIME OVER_(SYSTEM STOP)
   RUNG wire#powerrail
      Contact( "TIMING_MIN_DB".DONE )
      { S7_Templates := "time_type := Time" } "IEC_Timer_0_DB_80".TOF(pt := T#2S, et =>)
      wire#w1
      Coil( "ALARM DB PLC 2"."ORP-301 HIGH_SET VALIDATION TIME OVER_(SYSTEM STOP)" )
   END_RUNG
   RUNG wire#w1
      P_Trig( "P_TRIG".ARR[102] )
      S_Coil( "HOOTER" )
   END_RUNG
   // the same network as SCL:
   "IEC_Timer_0_DB_80".TOF(IN := "TIMING_MIN_DB".DONE, PT := T#2S);
   "ALARM DB PLC 2"."ORP-301 HIGH_SET VALIDATION TIME OVER_(SYSTEM STOP)" := "IEC_Timer_0_DB_80".Q;
   #_w1 := "IEC_Timer_0_DB_80".Q AND NOT "P_TRIG".ARR[102];   // rising edge
   "P_TRIG".ARR[102] := "IEC_Timer_0_DB_80".Q;
   IF #_w1 THEN "HOOTER" := TRUE; END_IF;
END_REGION

REGION Network 104: EDI-501A FEED PRESSURE FIT-501 LOW
   RUNG wire#powerrail
      { S7_Templates := "SrcType := Int" } EQ_Contact(in1 := "INTERLOCK DB"."EDI PARAMETER BUFF"."FIT-501 LOW BUFF", in2 := 2)
      wire#w1
      Coil( "ALARM DB PLC 2"."EDI-501A FEED PRESSURE FIT-501 LOW" )
   END_RUNG
   RUNG wire#w1
      P_Trig( "P_TRIG".ARR[103] )
      S_Coil( "HOOTER" )
   END_RUNG
   // the same network as SCL:
   "ALARM DB PLC 2"."EDI-501A FEED PRESSURE FIT-501 LOW" := "INTERLOCK DB"."EDI PARAMETER BUFF"."FIT-501 LOW BUFF" = 2;
   #_w1 := "ALARM DB PLC 2"."EDI-501A FEED PRESSURE FIT-501 LOW" AND NOT "P_TRIG".ARR[103];   // rising edge
   "P_TRIG".ARR[103] := "ALARM DB PLC 2"."EDI-501A FEED PRESSURE FIT-501 LOW";
   IF #_w1 THEN "HOOTER" := TRUE; END_IF;
END_REGION

REGION Network 105: FIT-501 LOW_SET VALIDATION TIME OVER_(SYSTEM STOP)
   RUNG wire#powerrail
      Contact( "TIMING_SECS_DB_16".DONE )
      { S7_Templates := "time_type := Time" } "IEC_Timer_0_DB_151".TOF(pt := T#2S, et =>)
      wire#w1
      Coil( "ALARM DB PLC 2"."FIT-501  LOW_SET VALIDATION TIME OVER_(SYSTEM STOP)" )
   END_RUNG
   RUNG wire#w1
      P_Trig( "P_TRIG".ARR[104] )
      S_Coil( "HOOTER" )
   END_RUNG
   // the same network as SCL:
   "IEC_Timer_0_DB_151".TOF(IN := "TIMING_SECS_DB_16".DONE, PT := T#2S);
   "ALARM DB PLC 2"."FIT-501  LOW_SET VALIDATION TIME OVER_(SYSTEM STOP)" := "IEC_Timer_0_DB_151".Q;
   #_w1 := "IEC_Timer_0_DB_151".Q AND NOT "P_TRIG".ARR[104];   // rising edge
   "P_TRIG".ARR[104] := "IEC_Timer_0_DB_151".Q;
   IF #_w1 THEN "HOOTER" := TRUE; END_IF;
END_REGION

REGION Network 106: EDI-501B FEED PRESSURE FIT-502 LOW
   RUNG wire#powerrail
      { S7_Templates := "SrcType := Int" } EQ_Contact(in1 := "INTERLOCK DB"."EDI PARAMETER BUFF"."FIT-502 LOW  BUFF", in2 := 2)
      wire#w1
      Coil( "ALARM DB PLC 2"."EDI-501B FEED PRESSURE FIT-502 LOW" )
   END_RUNG
   RUNG wire#w1
      P_Trig( "P_TRIG".ARR[105] )
      S_Coil( "HOOTER" )
   END_RUNG
   // the same network as SCL:
   "ALARM DB PLC 2"."EDI-501B FEED PRESSURE FIT-502 LOW" := "INTERLOCK DB"."EDI PARAMETER BUFF"."FIT-502 LOW  BUFF" = 2;
   #_w1 := "ALARM DB PLC 2"."EDI-501B FEED PRESSURE FIT-502 LOW" AND NOT "P_TRIG".ARR[105];   // rising edge
   "P_TRIG".ARR[105] := "ALARM DB PLC 2"."EDI-501B FEED PRESSURE FIT-502 LOW";
   IF #_w1 THEN "HOOTER" := TRUE; END_IF;
END_REGION

REGION Network 107: FIT-502 LOW_SET VALIDATION TIME OVER_(SYSTEM STOP)
   RUNG wire#powerrail
      Contact( "TIMING_SECS_DB_19".DONE )
      { S7_Templates := "time_type := Time" } "IEC_Timer_0_DB_152".TOF(pt := T#2S, et =>)
      wire#w1
      Coil( "ALARM DB PLC 2"."FIT-501 LOW_SET VALIDATION TIME OVER_(SYSTEM STOP)" )
   END_RUNG
   RUNG wire#w1
      P_Trig( "P_TRIG".ARR[106] )
      S_Coil( "HOOTER" )
   END_RUNG
   // the same network as SCL:
   "IEC_Timer_0_DB_152".TOF(IN := "TIMING_SECS_DB_19".DONE, PT := T#2S);
   "ALARM DB PLC 2"."FIT-501 LOW_SET VALIDATION TIME OVER_(SYSTEM STOP)" := "IEC_Timer_0_DB_152".Q;
   #_w1 := "IEC_Timer_0_DB_152".Q AND NOT "P_TRIG".ARR[106];   // rising edge
   "P_TRIG".ARR[106] := "IEC_Timer_0_DB_152".Q;
   IF #_w1 THEN "HOOTER" := TRUE; END_IF;
END_REGION

REGION Network 108: EDI-501B CONCENTRATE OUT PRESSURE FIT-503 LOW
   RUNG wire#powerrail
      { S7_Templates := "SrcType := Int" } EQ_Contact(in1 := "INTERLOCK DB"."EDI PARAMETER BUFF"."FIT-503 LOW BUFF", in2 := 2)
      wire#w1
      Coil( "ALARM DB PLC 2"."EDI-501B CONCENTRATE OUT PRESSURE FIT-503 LOW" )
   END_RUNG
   RUNG wire#w1
      P_Trig( "P_TRIG".ARR[107] )
      S_Coil( "HOOTER" )
   END_RUNG
   // the same network as SCL:
   "ALARM DB PLC 2"."EDI-501B CONCENTRATE OUT PRESSURE FIT-503 LOW" := "INTERLOCK DB"."EDI PARAMETER BUFF"."FIT-503 LOW BUFF" = 2;
   #_w1 := "ALARM DB PLC 2"."EDI-501B CONCENTRATE OUT PRESSURE FIT-503 LOW" AND NOT "P_TRIG".ARR[107];   // rising edge
   "P_TRIG".ARR[107] := "ALARM DB PLC 2"."EDI-501B CONCENTRATE OUT PRESSURE FIT-503 LOW";
   IF #_w1 THEN "HOOTER" := TRUE; END_IF;
END_REGION

REGION Network 109: FIT-503 LOW_SET VALIDATION TIME OVER_(SYSTEM STOP)
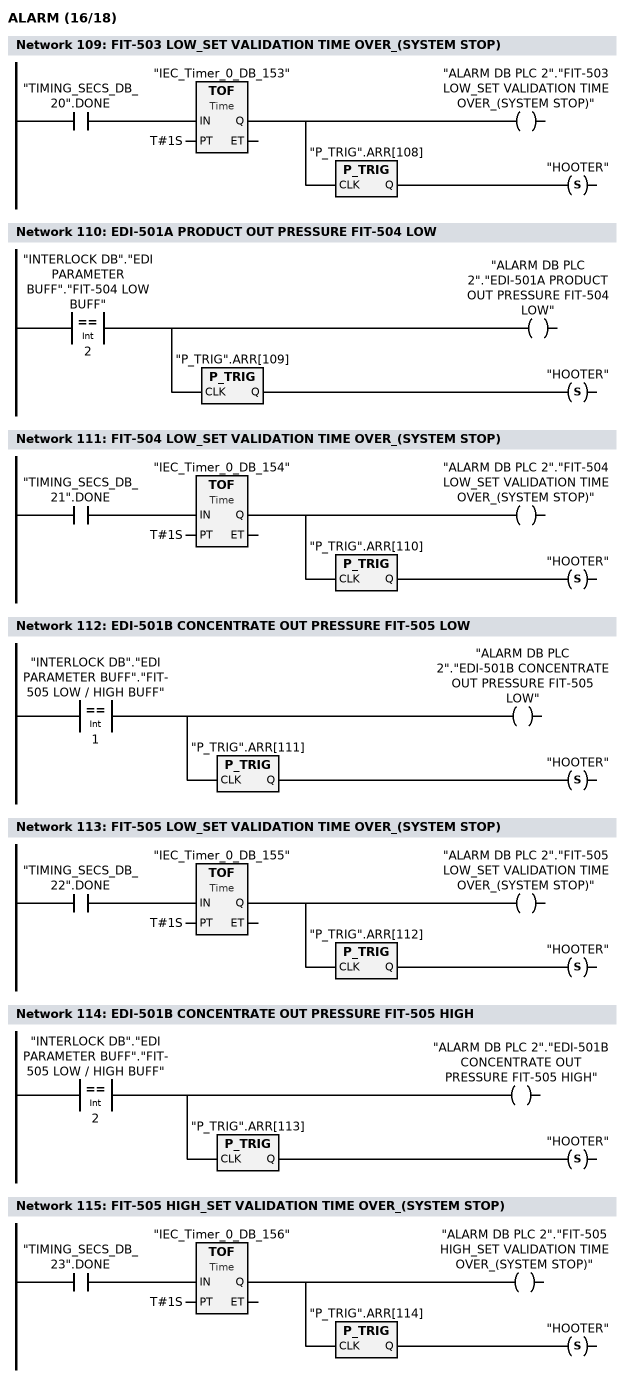
   RUNG wire#powerrail
      Contact( "TIMING_SECS_DB_20".DONE )
      { S7_Templates := "time_type := Time" } "IEC_Timer_0_DB_153".TOF(pt := T#1S, et =>)
      wire#w1
      Coil( "ALARM DB PLC 2"."FIT-503 LOW_SET VALIDATION TIME OVER_(SYSTEM STOP)" )
   END_RUNG
   RUNG wire#w1
      P_Trig( "P_TRIG".ARR[108] )
      S_Coil( "HOOTER" )
   END_RUNG
   // the same network as SCL:
   "IEC_Timer_0_DB_153".TOF(IN := "TIMING_SECS_DB_20".DONE, PT := T#1S);
   "ALARM DB PLC 2"."FIT-503 LOW_SET VALIDATION TIME OVER_(SYSTEM STOP)" := "IEC_Timer_0_DB_153".Q;
   #_w1 := "IEC_Timer_0_DB_153".Q AND NOT "P_TRIG".ARR[108];   // rising edge
   "P_TRIG".ARR[108] := "IEC_Timer_0_DB_153".Q;
   IF #_w1 THEN "HOOTER" := TRUE; END_IF;
END_REGION

REGION Network 110: EDI-501A PRODUCT OUT PRESSURE FIT-504 LOW
   RUNG wire#powerrail
      { S7_Templates := "SrcType := Int" } EQ_Contact(in1 := "INTERLOCK DB"."EDI PARAMETER BUFF"."FIT-504 LOW BUFF", in2 := 2)
      wire#w1
      Coil( "ALARM DB PLC 2"."EDI-501A PRODUCT OUT PRESSURE FIT-504 LOW" )
   END_RUNG
   RUNG wire#w1
      P_Trig( "P_TRIG".ARR[109] )
      S_Coil( "HOOTER" )
   END_RUNG
   // the same network as SCL:
   "ALARM DB PLC 2"."EDI-501A PRODUCT OUT PRESSURE FIT-504 LOW" := "INTERLOCK DB"."EDI PARAMETER BUFF"."FIT-504 LOW BUFF" = 2;
   #_w1 := "ALARM DB PLC 2"."EDI-501A PRODUCT OUT PRESSURE FIT-504 LOW" AND NOT "P_TRIG".ARR[109];   // rising edge
   "P_TRIG".ARR[109] := "ALARM DB PLC 2"."EDI-501A PRODUCT OUT PRESSURE FIT-504 LOW";
   IF #_w1 THEN "HOOTER" := TRUE; END_IF;
END_REGION

REGION Network 111: FIT-504 LOW_SET VALIDATION TIME OVER_(SYSTEM STOP)
   RUNG wire#powerrail
      Contact( "TIMING_SECS_DB_21".DONE )
      { S7_Templates := "time_type := Time" } "IEC_Timer_0_DB_154".TOF(pt := T#1S, et =>)
      wire#w1
      Coil( "ALARM DB PLC 2"."FIT-504 LOW_SET VALIDATION TIME OVER_(SYSTEM STOP)" )
   END_RUNG
   RUNG wire#w1
      P_Trig( "P_TRIG".ARR[110] )
      S_Coil( "HOOTER" )
   END_RUNG
   // the same network as SCL:
   "IEC_Timer_0_DB_154".TOF(IN := "TIMING_SECS_DB_21".DONE, PT := T#1S);
   "ALARM DB PLC 2"."FIT-504 LOW_SET VALIDATION TIME OVER_(SYSTEM STOP)" := "IEC_Timer_0_DB_154".Q;
   #_w1 := "IEC_Timer_0_DB_154".Q AND NOT "P_TRIG".ARR[110];   // rising edge
   "P_TRIG".ARR[110] := "IEC_Timer_0_DB_154".Q;
   IF #_w1 THEN "HOOTER" := TRUE; END_IF;
END_REGION

REGION Network 112: EDI-501B CONCENTRATE OUT PRESSURE FIT-505 LOW
   RUNG wire#powerrail
      { S7_Templates := "SrcType := Int" } EQ_Contact(in1 := "INTERLOCK DB"."EDI PARAMETER BUFF"."FIT-505 LOW / HIGH BUFF", in2 := 1)
      wire#w1
      Coil( "ALARM DB PLC 2"."EDI-501B CONCENTRATE OUT PRESSURE FIT-505 LOW" )
   END_RUNG
   RUNG wire#w1
      P_Trig( "P_TRIG".ARR[111] )
      S_Coil( "HOOTER" )
   END_RUNG
   // the same network as SCL:
   "ALARM DB PLC 2"."EDI-501B CONCENTRATE OUT PRESSURE FIT-505 LOW" := "INTERLOCK DB"."EDI PARAMETER BUFF"."FIT-505 LOW / HIGH BUFF" = 1;
   #_w1 := "ALARM DB PLC 2"."EDI-501B CONCENTRATE OUT PRESSURE FIT-505 LOW" AND NOT "P_TRIG".ARR[111];   // rising edge
   "P_TRIG".ARR[111] := "ALARM DB PLC 2"."EDI-501B CONCENTRATE OUT PRESSURE FIT-505 LOW";
   IF #_w1 THEN "HOOTER" := TRUE; END_IF;
END_REGION

REGION Network 113: FIT-505 LOW_SET VALIDATION TIME OVER_(SYSTEM STOP)
   RUNG wire#powerrail
      Contact( "TIMING_SECS_DB_22".DONE )
      { S7_Templates := "time_type := Time" } "IEC_Timer_0_DB_155".TOF(pt := T#1S, et =>)
      wire#w1
      Coil( "ALARM DB PLC 2"."FIT-505 LOW_SET VALIDATION TIME OVER_(SYSTEM STOP)" )
   END_RUNG
   RUNG wire#w1
      P_Trig( "P_TRIG".ARR[112] )
      S_Coil( "HOOTER" )
   END_RUNG
   // the same network as SCL:
   "IEC_Timer_0_DB_155".TOF(IN := "TIMING_SECS_DB_22".DONE, PT := T#1S);
   "ALARM DB PLC 2"."FIT-505 LOW_SET VALIDATION TIME OVER_(SYSTEM STOP)" := "IEC_Timer_0_DB_155".Q;
   #_w1 := "IEC_Timer_0_DB_155".Q AND NOT "P_TRIG".ARR[112];   // rising edge
   "P_TRIG".ARR[112] := "IEC_Timer_0_DB_155".Q;
   IF #_w1 THEN "HOOTER" := TRUE; END_IF;
END_REGION

REGION Network 114: EDI-501B CONCENTRATE OUT PRESSURE FIT-505 HIGH
   RUNG wire#powerrail
      { S7_Templates := "SrcType := Int" } EQ_Contact(in1 := "INTERLOCK DB"."EDI PARAMETER BUFF"."FIT-505 LOW / HIGH BUFF", in2 := 2)
      wire#w1
      Coil( "ALARM DB PLC 2"."EDI-501B CONCENTRATE OUT PRESSURE FIT-505 HIGH" )
   END_RUNG
   RUNG wire#w1
      P_Trig( "P_TRIG".ARR[113] )
      S_Coil( "HOOTER" )
   END_RUNG
   // the same network as SCL:
   "ALARM DB PLC 2"."EDI-501B CONCENTRATE OUT PRESSURE FIT-505 HIGH" := "INTERLOCK DB"."EDI PARAMETER BUFF"."FIT-505 LOW / HIGH BUFF" = 2;
   #_w1 := "ALARM DB PLC 2"."EDI-501B CONCENTRATE OUT PRESSURE FIT-505 HIGH" AND NOT "P_TRIG".ARR[113];   // rising edge
   "P_TRIG".ARR[113] := "ALARM DB PLC 2"."EDI-501B CONCENTRATE OUT PRESSURE FIT-505 HIGH";
   IF #_w1 THEN "HOOTER" := TRUE; END_IF;
END_REGION

REGION Network 115: FIT-505 HIGH_SET VALIDATION TIME OVER_(SYSTEM STOP)
   RUNG wire#powerrail
      Contact( "TIMING_SECS_DB_23".DONE )
      { S7_Templates := "time_type := Time" } "IEC_Timer_0_DB_156".TOF(pt := T#1S, et =>)
      wire#w1
      Coil( "ALARM DB PLC 2"."FIT-505 HIGH_SET VALIDATION TIME OVER_(SYSTEM STOP)" )
   END_RUNG
   RUNG wire#w1
      P_Trig( "P_TRIG".ARR[114] )
      S_Coil( "HOOTER" )
   END_RUNG
   // the same network as SCL:
   "IEC_Timer_0_DB_156".TOF(IN := "TIMING_SECS_DB_23".DONE, PT := T#1S);
   "ALARM DB PLC 2"."FIT-505 HIGH_SET VALIDATION TIME OVER_(SYSTEM STOP)" := "IEC_Timer_0_DB_156".Q;
   #_w1 := "IEC_Timer_0_DB_156".Q AND NOT "P_TRIG".ARR[114];   // rising edge
   "P_TRIG".ARR[114] := "IEC_Timer_0_DB_156".Q;
   IF #_w1 THEN "HOOTER" := TRUE; END_IF;
END_REGION

REGION Network 116: EDI-501A PRODUCT OUT PRESSURE FIT-506 LOW
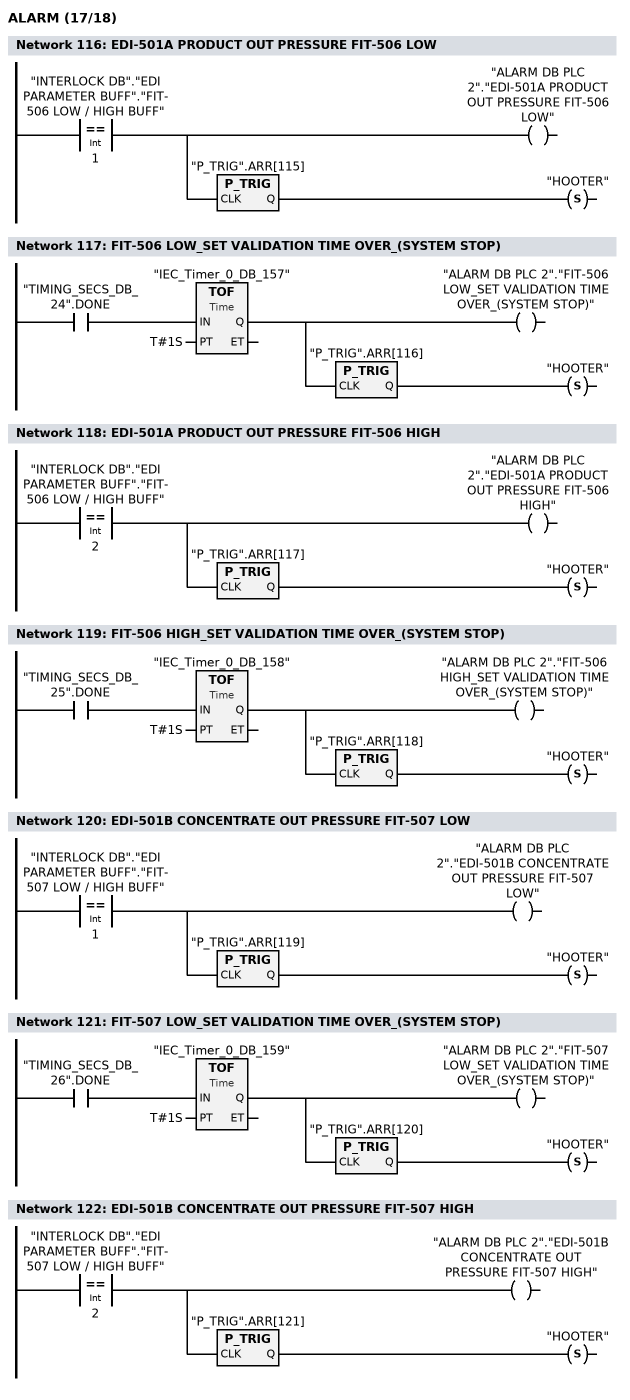
   RUNG wire#powerrail
      { S7_Templates := "SrcType := Int" } EQ_Contact(in1 := "INTERLOCK DB"."EDI PARAMETER BUFF"."FIT-506 LOW / HIGH BUFF", in2 := 1)
      wire#w1
      Coil( "ALARM DB PLC 2"."EDI-501A PRODUCT OUT PRESSURE FIT-506 LOW" )
   END_RUNG
   RUNG wire#w1
      P_Trig( "P_TRIG".ARR[115] )
      S_Coil( "HOOTER" )
   END_RUNG
   // the same network as SCL:
   "ALARM DB PLC 2"."EDI-501A PRODUCT OUT PRESSURE FIT-506 LOW" := "INTERLOCK DB"."EDI PARAMETER BUFF"."FIT-506 LOW / HIGH BUFF" = 1;
   #_w1 := "ALARM DB PLC 2"."EDI-501A PRODUCT OUT PRESSURE FIT-506 LOW" AND NOT "P_TRIG".ARR[115];   // rising edge
   "P_TRIG".ARR[115] := "ALARM DB PLC 2"."EDI-501A PRODUCT OUT PRESSURE FIT-506 LOW";
   IF #_w1 THEN "HOOTER" := TRUE; END_IF;
END_REGION

REGION Network 117: FIT-506 LOW_SET VALIDATION TIME OVER_(SYSTEM STOP)
   RUNG wire#powerrail
      Contact( "TIMING_SECS_DB_24".DONE )
      { S7_Templates := "time_type := Time" } "IEC_Timer_0_DB_157".TOF(pt := T#1S, et =>)
      wire#w1
      Coil( "ALARM DB PLC 2"."FIT-506 LOW_SET VALIDATION TIME OVER_(SYSTEM STOP)" )
   END_RUNG
   RUNG wire#w1
      P_Trig( "P_TRIG".ARR[116] )
      S_Coil( "HOOTER" )
   END_RUNG
   // the same network as SCL:
   "IEC_Timer_0_DB_157".TOF(IN := "TIMING_SECS_DB_24".DONE, PT := T#1S);
   "ALARM DB PLC 2"."FIT-506 LOW_SET VALIDATION TIME OVER_(SYSTEM STOP)" := "IEC_Timer_0_DB_157".Q;
   #_w1 := "IEC_Timer_0_DB_157".Q AND NOT "P_TRIG".ARR[116];   // rising edge
   "P_TRIG".ARR[116] := "IEC_Timer_0_DB_157".Q;
   IF #_w1 THEN "HOOTER" := TRUE; END_IF;
END_REGION

REGION Network 118: EDI-501A PRODUCT OUT PRESSURE FIT-506 HIGH
   RUNG wire#powerrail
      { S7_Templates := "SrcType := Int" } EQ_Contact(in1 := "INTERLOCK DB"."EDI PARAMETER BUFF"."FIT-506 LOW / HIGH BUFF", in2 := 2)
      wire#w1
      Coil( "ALARM DB PLC 2"."EDI-501A PRODUCT OUT PRESSURE FIT-506 HIGH" )
   END_RUNG
   RUNG wire#w1
      P_Trig( "P_TRIG".ARR[117] )
      S_Coil( "HOOTER" )
   END_RUNG
   // the same network as SCL:
   "ALARM DB PLC 2"."EDI-501A PRODUCT OUT PRESSURE FIT-506 HIGH" := "INTERLOCK DB"."EDI PARAMETER BUFF"."FIT-506 LOW / HIGH BUFF" = 2;
   #_w1 := "ALARM DB PLC 2"."EDI-501A PRODUCT OUT PRESSURE FIT-506 HIGH" AND NOT "P_TRIG".ARR[117];   // rising edge
   "P_TRIG".ARR[117] := "ALARM DB PLC 2"."EDI-501A PRODUCT OUT PRESSURE FIT-506 HIGH";
   IF #_w1 THEN "HOOTER" := TRUE; END_IF;
END_REGION

REGION Network 119: FIT-506 HIGH_SET VALIDATION TIME OVER_(SYSTEM STOP)
   RUNG wire#powerrail
      Contact( "TIMING_SECS_DB_25".DONE )
      { S7_Templates := "time_type := Time" } "IEC_Timer_0_DB_158".TOF(pt := T#1S, et =>)
      wire#w1
      Coil( "ALARM DB PLC 2"."FIT-506 HIGH_SET VALIDATION TIME OVER_(SYSTEM STOP)" )
   END_RUNG
   RUNG wire#w1
      P_Trig( "P_TRIG".ARR[118] )
      S_Coil( "HOOTER" )
   END_RUNG
   // the same network as SCL:
   "IEC_Timer_0_DB_158".TOF(IN := "TIMING_SECS_DB_25".DONE, PT := T#1S);
   "ALARM DB PLC 2"."FIT-506 HIGH_SET VALIDATION TIME OVER_(SYSTEM STOP)" := "IEC_Timer_0_DB_158".Q;
   #_w1 := "IEC_Timer_0_DB_158".Q AND NOT "P_TRIG".ARR[118];   // rising edge
   "P_TRIG".ARR[118] := "IEC_Timer_0_DB_158".Q;
   IF #_w1 THEN "HOOTER" := TRUE; END_IF;
END_REGION

REGION Network 120: EDI-501B CONCENTRATE OUT PRESSURE FIT-507 LOW
   RUNG wire#powerrail
      { S7_Templates := "SrcType := Int" } EQ_Contact(in1 := "INTERLOCK DB"."EDI PARAMETER BUFF"."FIT-507 LOW / HIGH BUFF", in2 := 1)
      wire#w1
      Coil( "ALARM DB PLC 2"."EDI-501B CONCENTRATE OUT PRESSURE FIT-507 LOW" )
   END_RUNG
   RUNG wire#w1
      P_Trig( "P_TRIG".ARR[119] )
      S_Coil( "HOOTER" )
   END_RUNG
   // the same network as SCL:
   "ALARM DB PLC 2"."EDI-501B CONCENTRATE OUT PRESSURE FIT-507 LOW" := "INTERLOCK DB"."EDI PARAMETER BUFF"."FIT-507 LOW / HIGH BUFF" = 1;
   #_w1 := "ALARM DB PLC 2"."EDI-501B CONCENTRATE OUT PRESSURE FIT-507 LOW" AND NOT "P_TRIG".ARR[119];   // rising edge
   "P_TRIG".ARR[119] := "ALARM DB PLC 2"."EDI-501B CONCENTRATE OUT PRESSURE FIT-507 LOW";
   IF #_w1 THEN "HOOTER" := TRUE; END_IF;
END_REGION

REGION Network 121: FIT-507 LOW_SET VALIDATION TIME OVER_(SYSTEM STOP)
   RUNG wire#powerrail
      Contact( "TIMING_SECS_DB_26".DONE )
      { S7_Templates := "time_type := Time" } "IEC_Timer_0_DB_159".TOF(pt := T#1S, et =>)
      wire#w1
      Coil( "ALARM DB PLC 2"."FIT-507 LOW_SET VALIDATION TIME OVER_(SYSTEM STOP)" )
   END_RUNG
   RUNG wire#w1
      P_Trig( "P_TRIG".ARR[120] )
      S_Coil( "HOOTER" )
   END_RUNG
   // the same network as SCL:
   "IEC_Timer_0_DB_159".TOF(IN := "TIMING_SECS_DB_26".DONE, PT := T#1S);
   "ALARM DB PLC 2"."FIT-507 LOW_SET VALIDATION TIME OVER_(SYSTEM STOP)" := "IEC_Timer_0_DB_159".Q;
   #_w1 := "IEC_Timer_0_DB_159".Q AND NOT "P_TRIG".ARR[120];   // rising edge
   "P_TRIG".ARR[120] := "IEC_Timer_0_DB_159".Q;
   IF #_w1 THEN "HOOTER" := TRUE; END_IF;
END_REGION

REGION Network 122: EDI-501B CONCENTRATE OUT PRESSURE FIT-507 HIGH
   RUNG wire#powerrail
      { S7_Templates := "SrcType := Int" } EQ_Contact(in1 := "INTERLOCK DB"."EDI PARAMETER BUFF"."FIT-507 LOW / HIGH BUFF", in2 := 2)
      wire#w1
      Coil( "ALARM DB PLC 2"."EDI-501B CONCENTRATE OUT PRESSURE FIT-507 HIGH" )
   END_RUNG
   RUNG wire#w1
      P_Trig( "P_TRIG".ARR[121] )
      S_Coil( "HOOTER" )
   END_RUNG
   // the same network as SCL:
   "ALARM DB PLC 2"."EDI-501B CONCENTRATE OUT PRESSURE FIT-507 HIGH" := "INTERLOCK DB"."EDI PARAMETER BUFF"."FIT-507 LOW / HIGH BUFF" = 2;
   #_w1 := "ALARM DB PLC 2"."EDI-501B CONCENTRATE OUT PRESSURE FIT-507 HIGH" AND NOT "P_TRIG".ARR[121];   // rising edge
   "P_TRIG".ARR[121] := "ALARM DB PLC 2"."EDI-501B CONCENTRATE OUT PRESSURE FIT-507 HIGH";
   IF #_w1 THEN "HOOTER" := TRUE; END_IF;
END_REGION

REGION Network 123: FIT-507 HIGH_SET VALIDATION TIME OVER_(SYSTEM STOP)
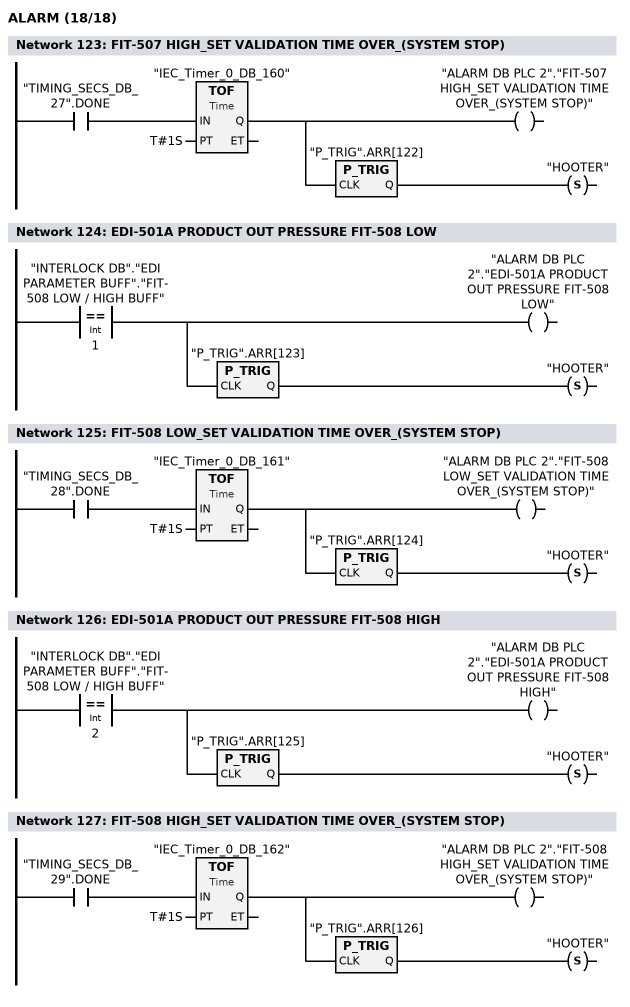
   RUNG wire#powerrail
      Contact( "TIMING_SECS_DB_27".DONE )
      { S7_Templates := "time_type := Time" } "IEC_Timer_0_DB_160".TOF(pt := T#1S, et =>)
      wire#w1
      Coil( "ALARM DB PLC 2"."FIT-507 HIGH_SET VALIDATION TIME OVER_(SYSTEM STOP)" )
   END_RUNG
   RUNG wire#w1
      P_Trig( "P_TRIG".ARR[122] )
      S_Coil( "HOOTER" )
   END_RUNG
   // the same network as SCL:
   "IEC_Timer_0_DB_160".TOF(IN := "TIMING_SECS_DB_27".DONE, PT := T#1S);
   "ALARM DB PLC 2"."FIT-507 HIGH_SET VALIDATION TIME OVER_(SYSTEM STOP)" := "IEC_Timer_0_DB_160".Q;
   #_w1 := "IEC_Timer_0_DB_160".Q AND NOT "P_TRIG".ARR[122];   // rising edge
   "P_TRIG".ARR[122] := "IEC_Timer_0_DB_160".Q;
   IF #_w1 THEN "HOOTER" := TRUE; END_IF;
END_REGION

REGION Network 124: EDI-501A PRODUCT OUT PRESSURE FIT-508 LOW
   RUNG wire#powerrail
      { S7_Templates := "SrcType := Int" } EQ_Contact(in1 := "INTERLOCK DB"."EDI PARAMETER BUFF"."FIT-508 LOW / HIGH BUFF", in2 := 1)
      wire#w1
      Coil( "ALARM DB PLC 2"."EDI-501A PRODUCT OUT PRESSURE FIT-508 LOW" )
   END_RUNG
   RUNG wire#w1
      P_Trig( "P_TRIG".ARR[123] )
      S_Coil( "HOOTER" )
   END_RUNG
   // the same network as SCL:
   "ALARM DB PLC 2"."EDI-501A PRODUCT OUT PRESSURE FIT-508 LOW" := "INTERLOCK DB"."EDI PARAMETER BUFF"."FIT-508 LOW / HIGH BUFF" = 1;
   #_w1 := "ALARM DB PLC 2"."EDI-501A PRODUCT OUT PRESSURE FIT-508 LOW" AND NOT "P_TRIG".ARR[123];   // rising edge
   "P_TRIG".ARR[123] := "ALARM DB PLC 2"."EDI-501A PRODUCT OUT PRESSURE FIT-508 LOW";
   IF #_w1 THEN "HOOTER" := TRUE; END_IF;
END_REGION

REGION Network 125: FIT-508 LOW_SET VALIDATION TIME OVER_(SYSTEM STOP)
   RUNG wire#powerrail
      Contact( "TIMING_SECS_DB_28".DONE )
      { S7_Templates := "time_type := Time" } "IEC_Timer_0_DB_161".TOF(pt := T#1S, et =>)
      wire#w1
      Coil( "ALARM DB PLC 2"."FIT-508 LOW_SET VALIDATION TIME OVER_(SYSTEM STOP)" )
   END_RUNG
   RUNG wire#w1
      P_Trig( "P_TRIG".ARR[124] )
      S_Coil( "HOOTER" )
   END_RUNG
   // the same network as SCL:
   "IEC_Timer_0_DB_161".TOF(IN := "TIMING_SECS_DB_28".DONE, PT := T#1S);
   "ALARM DB PLC 2"."FIT-508 LOW_SET VALIDATION TIME OVER_(SYSTEM STOP)" := "IEC_Timer_0_DB_161".Q;
   #_w1 := "IEC_Timer_0_DB_161".Q AND NOT "P_TRIG".ARR[124];   // rising edge
   "P_TRIG".ARR[124] := "IEC_Timer_0_DB_161".Q;
   IF #_w1 THEN "HOOTER" := TRUE; END_IF;
END_REGION

REGION Network 126: EDI-501A PRODUCT OUT PRESSURE FIT-508 HIGH
   RUNG wire#powerrail
      { S7_Templates := "SrcType := Int" } EQ_Contact(in1 := "INTERLOCK DB"."EDI PARAMETER BUFF"."FIT-508 LOW / HIGH BUFF", in2 := 2)
      wire#w1
      Coil( "ALARM DB PLC 2"."EDI-501A PRODUCT OUT PRESSURE FIT-508 HIGH" )
   END_RUNG
   RUNG wire#w1
      P_Trig( "P_TRIG".ARR[125] )
      S_Coil( "HOOTER" )
   END_RUNG
   // the same network as SCL:
   "ALARM DB PLC 2"."EDI-501A PRODUCT OUT PRESSURE FIT-508 HIGH" := "INTERLOCK DB"."EDI PARAMETER BUFF"."FIT-508 LOW / HIGH BUFF" = 2;
   #_w1 := "ALARM DB PLC 2"."EDI-501A PRODUCT OUT PRESSURE FIT-508 HIGH" AND NOT "P_TRIG".ARR[125];   // rising edge
   "P_TRIG".ARR[125] := "ALARM DB PLC 2"."EDI-501A PRODUCT OUT PRESSURE FIT-508 HIGH";
   IF #_w1 THEN "HOOTER" := TRUE; END_IF;
END_REGION

REGION Network 127: FIT-508 HIGH_SET VALIDATION TIME OVER_(SYSTEM STOP)
   RUNG wire#powerrail
      Contact( "TIMING_SECS_DB_29".DONE )
      { S7_Templates := "time_type := Time" } "IEC_Timer_0_DB_162".TOF(pt := T#1S, et =>)
      wire#w1
      Coil( "ALARM DB PLC 2"."FIT-508 HIGH_SET VALIDATION TIME OVER_(SYSTEM STOP)" )
   END_RUNG
   RUNG wire#w1
      P_Trig( "P_TRIG".ARR[126] )
      S_Coil( "HOOTER" )
   END_RUNG
   // the same network as SCL:
   "IEC_Timer_0_DB_162".TOF(IN := "TIMING_SECS_DB_29".DONE, PT := T#1S);
   "ALARM DB PLC 2"."FIT-508 HIGH_SET VALIDATION TIME OVER_(SYSTEM STOP)" := "IEC_Timer_0_DB_162".Q;
   #_w1 := "IEC_Timer_0_DB_162".Q AND NOT "P_TRIG".ARR[126];   // rising edge
   "P_TRIG".ARR[126] := "IEC_Timer_0_DB_162".Q;
   IF #_w1 THEN "HOOTER" := TRUE; END_IF;
END_REGION
END_FUNCTION
